C07273=1019.893,90.368,388.919,167.159,51.972,159.571
C07274=1019.887,90.119,388.936,167.157,51.979,159.572
C07275=1019.882,89.870,388.955,167.154,51.985,159.572
C07276=1019.877,89.621,388.972,167.151,51.992,159.573
C07277=1019.872,89.371,388.989,167.149,51.999,159.574
C07278=1019.866,89.122,389.007,167.146,52.005,159.575
C07279=1019.860,88.872,389.025,167.143,52.012,159.575
C07280=1019.855,88.623,389.042,167.141,52.018,159.576
C07281=1019.849,88.374,389.059,167.139,52.025,159.577
C07282=1019.844,88.125,389.077,167.135,52.032,159.578
C07283=1019.838,87.875,389.094,167.133,52.039,159.579
C07284=1019.833,87.626,389.111,167.130,52.046,159.580
C07285=1019.828,87.377,389.129,167.127,52.052,159.580
C07286=1019.821,87.127,389.146,167.124,52.059,159.581
C07287=1019.816,86.877,389.163,167.122,52.065,159.582
C07288=1019.811,86.628,389.181,167.120,52.072,159.583
C07289=1019.805,86.379,389.198,167.116,52.079,159.583
C07290=1019.800,86.130,389.215,167.114,52.085,159.584
C07291=1019.794,85.881,389.233,167.111,52.092,159.585
C07292=1019.789,85.632,389.250,167.108,52.099,159.586
C07293=1019.784,85.382,389.267,167.106,52.106,159.587
C07294=1019.778,85.132,389.285,167.103,52.113,159.587
C07295=1019.772,84.882,389.302,167.100,52.119,159.588
C07296=1019.767,84.633,389.320,167.097,52.126,159.589
C07297=1019.761,84.384,389.337,167.095,52.132,159.590
C07298=1019.756,84.135,389.354,167.093,52.139,159.591
C07299=1019.751,83.886,389.372,167.089,52.145,159.591
C07300=1019.745,83.636,389.388,167.087,52.152,159.592
C07301=1019.739,83.387,389.405,167.085,52.159,159.593
C07302=1019.734,83.138,389.422,167.081,52.166,159.594
C07303=1019.728,82.889,389.440,167.079,52.172,159.594
C07304=1019.723,82.640,389.457,167.076,52.179,159.595
C07305=1019.718,82.390,389.474,167.073,52.185,159.596
C07306=1019.712,82.141,389.492,167.071,52.192,159.597
C07307=1019.706,81.891,389.509,167.068,52.198,159.597
C07308=1019.701,81.641,389.527,167.065,52.205,159.598
C07309=1019.696,81.392,389.543,167.063,52.212,159.599
C07310=1019.690,81.143,389.561,167.060,52.218,159.600
C07311=1019.685,80.893,389.578,167.057,52.225,159.601
C07312=1019.679,80.644,389.595,167.055,52.232,159.602
C07313=1019.674,80.394,389.612,167.052,52.239,159.602
C07314=1019.669,80.145,389.630,167.049,52.245,159.603
C07315=1019.663,79.896,389.647,167.047,52.251,159.604
C07316=1019.658,79.647,389.664,167.044,52.258,159.605
C07317=1019.653,79.397,389.681,167.041,52.264,159.605
C07318=1019.647,79.148,389.699,167.039,52.271,159.606
C07319=1019.641,78.899,389.715,167.036,52.278,159.607
C07320=1019.636,78.650,389.733,167.033,52.284,159.608
C07321=1019.630,78.400,389.749,167.031,52.291,159.608
C07322=1019.625,78.151,389.767,167.028,52.297,159.609
C07323=1019.620,77.901,389.784,167.026,52.304,159.610
C07324=1019.615,77.652,389.801,167.023,52.311,159.611
C07325=1019.609,77.403,389.818,167.021,52.317,159.611
C07326=1019.604,77.153,389.835,167.018,52.324,159.612
C07327=1019.598,76.904,389.853,167.015,52.330,159.613
C07328=1019.592,76.654,389.869,167.013,52.336,159.614
C07329=1019.587,76.405,389.886,167.010,52.343,159.615
C07330=1019.582,76.156,389.903,167.007,52.350,159.615
C07331=1019.576,75.906,389.920,167.004,52.357,159.616
C07332=1019.570,75.657,389.936,167.002,52.363,159.617
C07333=1019.564,75.374,389.955,166.999,52.371,159.618
C07334=1019.558,75.091,389.974,166.996,52.379,159.619
C07335=1019.552,74.810,389.994,166.993,52.386,159.620
C07336=1019.546,74.527,390.013,166.990,52.394,159.621
C07337=1019.541,74.277,390.030,166.987,52.401,159.621
C07338=1019.535,74.027,390.046,166.984,52.407,159.622
C07339=1019.530,73.778,390.063,166.982,52.413,159.623
C07340=1019.524,73.529,390.080,166.979,52.421,159.624
C07341=1019.519,73.279,390.097,166.977,52.427,159.624
C07342=1019.513,73.030,390.113,166.974,52.433,159.625
C07343=1019.508,72.780,390.130,166.971,52.440,159.626
C07344=1019.502,72.531,390.147,166.969,52.447,159.627
C07345=1019.496,72.282,390.164,166.965,52.453,159.627
C07346=1019.491,72.032,390.181,166.963,52.460,159.628
C07347=1019.486,71.783,390.198,166.961,52.467,159.629
C07348=1019.480,71.533,390.214,166.958,52.473,159.630
C07349=1019.475,71.284,390.230,166.955,52.480,159.631
C07350=1019.469,71.035,390.247,166.953,52.487,159.631
C07351=1019.464,70.786,390.264,166.950,52.493,159.632
C07352=1019.458,70.536,390.281,166.948,52.500,159.633
C07353=1019.453,70.287,390.297,166.945,52.507,159.634
C07354=1019.447,70.037,390.314,166.942,52.513,159.634
C07355=1019.442,69.788,390.331,166.940,52.520,159.635
C07356=1019.436,69.538,390.347,166.938,52.526,159.636
C07357=1019.431,69.289,390.364,166.934,52.533,159.637
C07358=1019.426,69.040,390.380,166.932,52.540,159.637
C07359=1019.420,68.790,390.397,166.930,52.546,159.638
C07360=1019.415,68.541,390.414,166.926,52.553,159.639
C07361=1019.409,68.292,390.431,166.924,52.559,159.640
C07362=1019.404,68.042,390.448,166.922,52.566,159.641
C07363=1019.398,67.793,390.464,166.918,52.573,159.641
C07364=1019.393,67.543,390.481,166.916,52.579,159.642
C07365=1019.387,67.295,390.497,166.914,52.586,159.643
C07366=1019.382,67.045,390.513,166.910,52.592,159.644
C07367=1019.376,66.796,390.530,166.908,52.599,159.644
C07368=1019.370,66.546,390.545,166.906,52.606,159.645
C07369=1019.365,66.296,390.562,166.903,52.612,159.646
C07370=1019.359,66.047,390.578,166.900,52.619,159.647
C07371=1019.355,65.798,390.595,166.898,52.626,159.648
C07372=1019.349,65.548,390.611,166.895,52.632,159.648
C07373=1019.343,65.299,390.628,166.893,52.639,159.649
C07374=1019.337,65.049,390.644,166.891,52.646,159.650
C07375=1019.332,64.800,390.661,166.887,52.653,159.651
C07376=1019.326,64.550,390.677,166.885,52.659,159.651
C07377=1019.321,64.302,390.693,166.882,52.666,159.652
C07378=1019.316,64.052,390.710,166.880,52.673,159.653
C07379=1019.310,63.803,390.726,166.877,52.679,159.654
C07380=1019.305,63.552,390.742,166.874,52.686,159.654
C07381=1019.299,63.303,390.759,166.871,52.692,159.655
C07382=1019.294,63.054,390.775,166.869,52.699,159.656
C07383=1019.288,62.805,390.791,166.866,52.706,159.657
C07384=1019.282,62.555,390.808,166.864,52.713,159.658
C07385=1019.277,62.305,390.823,166.860,52.719,159.658
C07386=1019.271,62.056,390.839,166.858,52.726,159.659
C07387=1019.265,61.807,390.855,166.856,52.733,159.660
C07388=1019.260,61.557,390.871,166.853,52.740,159.661
C07389=1019.254,61.308,390.887,166.851,52.746,159.662
C07390=1019.248,61.059,390.903,166.848,52.754,159.662
C07391=1019.243,60.808,390.920,166.845,52.760,159.663
C07392=1019.238,60.560,390.935,166.842,52.767,159.664
C07393=1019.232,60.310,390.952,166.840,52.774,159.665
C07394=1019.226,60.060,390.967,166.838,52.780,159.666
C07395=1019.220,59.811,390.984,166.835,52.787,159.666
C07396=1019.215,59.562,390.999,166.832,52.793,159.667
C07397=1019.208,59.279,391.017,166.830,52.801,159.668
C07398=1019.202,58.996,391.036,166.826,52.810,159.669
C07399=1019.195,58.713,391.054,166.823,52.817,159.670
C07400=1019.189,58.431,391.072,166.820,52.825,159.671
C07401=1019.184,58.181,391.088,166.818,52.831,159.672
C07402=1019.178,57.932,391.104,166.815,52.838,159.672
C07403=1019.172,57.682,391.120,166.812,52.845,159.673
C07404=1019.167,57.433,391.136,166.809,52.852,159.674
C07405=1019.161,57.184,391.152,166.807,52.858,159.675
C07406=1019.155,56.934,391.167,166.805,52.865,159.675
C07407=1019.150,56.685,391.183,166.802,52.872,159.676
C07408=1019.144,56.435,391.199,166.800,52.878,159.677
C07409=1019.139,56.186,391.215,166.796,52.885,159.677
C07410=1019.133,55.937,391.230,166.794,52.892,159.678
C07411=1019.128,55.687,391.246,166.792,52.898,159.679
C07412=1019.122,55.438,391.263,166.788,52.905,159.680
C07413=1019.117,55.188,391.278,166.786,52.912,159.681
C07414=1019.111,54.939,391.295,166.784,52.918,159.682
C07415=1019.106,54.689,391.310,166.781,52.925,159.682
C07416=1019.100,54.440,391.326,166.779,52.932,159.683
C07417=1019.095,54.190,391.342,166.775,52.939,159.684
C07418=1019.089,53.941,391.358,166.773,52.945,159.684
C07419=1019.084,53.692,391.373,166.771,52.952,159.685
C07420=1019.078,53.442,391.389,166.768,52.959,159.686
C07421=1019.072,53.193,391.405,166.765,52.965,159.687
C07422=1019.067,52.944,391.421,166.763,52.972,159.688
C07423=1019.061,52.694,391.436,166.760,52.979,159.688
C07424=1019.056,52.444,391.453,166.758,52.985,159.689
C07425=1019.051,52.195,391.468,166.755,52.992,159.690
C07426=1019.045,51.946,391.485,166.752,52.998,159.690
C07427=1019.039,51.696,391.500,166.750,53.005,159.691
C07428=1019.034,51.447,391.516,166.747,53.012,159.692
C07429=1019.028,51.197,391.532,166.744,53.018,159.693
C07430=1019.023,50.948,391.547,166.742,53.025,159.694
C07431=1019.017,50.698,391.563,166.739,53.032,159.694
C07432=1019.012,50.448,391.579,166.737,53.038,159.695
C07433=1019.006,50.200,391.594,166.735,53.045,159.696
C07434=1019.001,49.950,391.610,166.731,53.052,159.697
C07435=1018.995,49.701,391.626,166.729,53.058,159.697
C07436=1018.990,49.451,391.641,166.727,53.064,159.698
C07437=1018.985,49.201,391.658,166.724,53.072,159.699
C07438=1018.979,48.952,391.673,166.721,53.078,159.700
C07439=1018.974,48.702,391.689,166.719,53.085,159.700
C07440=1018.968,48.454,391.705,166.715,53.091,159.701
C07441=1018.963,48.204,391.720,166.713,53.098,159.702
C07442=1018.958,47.954,391.736,166.711,53.104,159.703
C07443=1018.952,47.705,391.752,166.708,53.111,159.703
C07444=1018.947,47.456,391.767,166.705,53.117,159.704
C07445=1018.941,47.206,391.783,166.703,53.124,159.705
C07446=1018.935,46.957,391.799,166.701,53.130,159.706
C07447=1018.930,46.707,391.814,166.698,53.137,159.706
C07448=1018.924,46.457,391.830,166.695,53.143,159.707
C07449=1018.919,46.209,391.845,166.693,53.150,159.708
C07450=1018.913,45.959,391.861,166.690,53.157,159.708
C07451=1018.908,45.709,391.876,166.688,53.164,159.709
C07452=1018.903,45.460,391.893,166.685,53.170,159.710
C07453=1018.898,45.210,391.908,166.682,53.177,159.711
C07454=1018.892,44.961,391.924,166.680,53.183,159.711
C07455=1018.887,44.712,391.940,166.678,53.190,159.712
C07456=1018.881,44.462,391.955,166.675,53.196,159.713
C07457=1018.876,44.213,391.970,166.672,53.202,159.713
C07458=1018.870,43.963,391.987,166.670,53.209,159.714
C07459=1018.865,43.714,392.002,166.667,53.215,159.715
C07460=1018.860,43.464,392.017,166.664,53.222,159.716
C07461=1018.854,43.182,392.035,166.661,53.230,159.717
C07462=1018.848,42.898,392.053,166.658,53.237,159.717
C07463=1018.842,42.616,392.070,166.655,53.244,159.718
C07464=1018.835,42.333,392.088,166.653,53.252,159.719
C07465=1018.830,42.083,392.103,166.650,53.258,159.720
C07466=1018.824,41.833,392.119,166.648,53.265,159.721
C07467=1018.819,41.584,392.134,166.644,53.271,159.721
C07468=1018.814,41.335,392.148,166.642,53.278,159.722
C07469=1018.808,41.085,392.164,166.640,53.284,159.723
C07470=1018.803,40.836,392.180,166.637,53.292,159.723
C07471=1018.797,40.586,392.195,166.635,53.298,159.724
C07472=1018.792,40.337,392.210,166.632,53.305,159.725
C07473=1018.786,40.088,392.225,166.629,53.312,159.726
C07474=1018.781,39.838,392.241,166.627,53.318,159.726
C07475=1018.775,39.588,392.256,166.624,53.325,159.727
C07476=1018.770,39.339,392.271,166.621,53.331,159.728
C07477=1018.763,39.089,392.286,166.619,53.338,159.729
C07478=1018.758,38.840,392.301,166.616,53.345,159.729
C07479=1018.753,38.591,392.317,166.614,53.351,159.730
C07480=1018.748,38.341,392.332,166.611,53.358,159.731
C07481=1018.742,38.092,392.347,166.608,53.365,159.732
C07482=1018.736,37.842,392.362,166.606,53.371,159.732
C07483=1018.731,37.593,392.377,166.604,53.378,159.733
C07484=1018.726,37.343,392.393,166.600,53.384,159.734
C07485=1018.721,37.093,392.408,166.598,53.391,159.735
C07486=1018.715,36.845,392.423,166.596,53.397,159.735
C07487=1018.709,36.595,392.438,166.593,53.404,159.736
C07488=1018.704,36.345,392.453,166.591,53.411,159.737
C07489=1018.698,36.096,392.468,166.587,53.418,159.738
C07490=1018.693,35.846,392.483,166.585,53.424,159.738
C07491=1018.687,35.597,392.497,166.583,53.431,159.739
C07492=1018.682,35.347,392.513,166.580,53.437,159.740
C07493=1018.676,35.098,392.528,166.578,53.444,159.741
C07494=1018.671,34.849,392.543,166.575,53.451,159.741
C07495=1018.664,34.599,392.558,166.572,53.458,159.742
C07496=1018.660,34.349,392.572,166.569,53.465,159.743
C07497=1018.653,34.099,392.587,166.567,53.471,159.743
C07498=1018.648,33.850,392.602,166.565,53.478,159.744
C07499=1018.642,33.601,392.617,166.561,53.484,159.745
C07500=1018.637,33.351,392.632,166.559,53.491,159.746
C07501=1018.631,33.102,392.646,166.556,53.498,159.746
C07502=1018.626,32.852,392.661,166.554,53.504,159.747
C07503=1018.620,32.603,392.676,166.552,53.511,159.748
C07504=1018.615,32.353,392.691,166.548,53.518,159.749
C07505=1018.609,32.104,392.705,166.546,53.525,159.749
C07506=1018.604,31.854,392.721,166.543,53.531,159.750
C07507=1018.598,31.605,392.735,166.541,53.538,159.751
C07508=1018.593,31.356,392.751,166.538,53.544,159.752
C07509=1018.588,31.105,392.765,166.535,53.552,159.752
C07510=1018.582,30.856,392.780,166.533,53.558,159.753
C07511=1018.577,30.607,392.795,166.530,53.565,159.754
C07512=1018.570,30.357,392.810,166.528,53.571,159.754
C07513=1018.566,30.107,392.825,166.525,53.577,159.755
C07514=1018.560,29.858,392.839,166.522,53.584,159.756
C07515=1018.555,29.609,392.854,166.520,53.591,159.757
C07516=1018.549,29.359,392.869,166.518,53.598,159.757
C07517=1018.544,29.110,392.884,166.514,53.604,159.758
C07518=1018.538,28.861,392.898,166.512,53.611,159.759
C07519=1018.532,28.610,392.913,166.509,53.617,159.759
C07520=1018.527,28.361,392.928,166.507,53.624,159.760
C07521=1018.522,28.112,392.943,166.505,53.630,159.761
C07522=1018.516,27.862,392.957,166.501,53.637,159.761
C07523=1018.511,27.612,392.972,166.499,53.644,159.762
C07524=1018.505,27.363,392.987,166.497,53.650,159.763
C07525=1018.499,27.089,393.003,166.494,53.658,159.764
C07526=1018.492,26.814,393.019,166.491,53.665,159.765
C07527=1018.486,26.539,393.035,166.488,53.673,159.766
C07528=1018.480,26.265,393.051,166.485,53.680,159.766
C07529=1018.475,26.007,393.065,166.482,53.687,159.767
C07530=1018.469,25.749,393.081,166.479,53.694,159.768
C07531=1018.463,25.491,393.096,166.477,53.701,159.769
C07532=1018.457,25.233,393.110,166.474,53.708,159.769
C07533=1018.452,24.984,393.125,166.471,53.714,159.770
C07534=1018.447,24.734,393.139,166.468,53.721,159.771
C07535=1018.441,24.485,393.154,166.466,53.727,159.771
C07536=1018.435,24.235,393.168,166.463,53.735,159.772
C07537=1018.430,23.985,393.183,166.461,53.741,159.773
C07538=1018.424,23.736,393.197,166.459,53.748,159.774
C07539=1018.419,23.487,393.212,166.455,53.754,159.774
C07540=1018.413,23.237,393.226,166.453,53.761,159.775
C07541=1018.408,22.987,393.240,166.450,53.768,159.776
C07542=1018.402,22.738,393.255,166.448,53.775,159.777
C07543=1018.397,22.488,393.269,166.444,53.781,159.777
C07544=1018.391,22.239,393.283,166.443,53.788,159.778
C07545=1018.386,21.989,393.298,166.440,53.794,159.779
C07546=1018.380,21.739,393.312,166.437,53.802,159.779
C07547=1018.374,21.490,393.327,166.435,53.808,159.780
C07548=1018.369,21.241,393.341,166.431,53.814,159.781
C07549=1018.364,20.991,393.356,166.429,53.821,159.782
C07550=1018.358,20.742,393.370,166.427,53.827,159.782
C07551=1018.353,20.492,393.384,166.424,53.835,159.783
C07552=1018.347,20.243,393.398,166.422,53.841,159.784
C07553=1018.342,19.993,393.413,166.419,53.848,159.784
C07554=1018.336,19.743,393.427,166.416,53.854,159.785
C07555=1018.330,19.494,393.441,166.414,53.860,159.786
C07556=1018.325,19.245,393.455,166.411,53.868,159.786
C07557=1018.320,18.995,393.470,166.409,53.874,159.787
C07558=1018.314,18.746,393.484,166.406,53.881,159.788
C07559=1018.309,18.496,393.498,166.403,53.887,159.789
C07560=1018.303,18.246,393.512,166.400,53.894,159.789
C07561=1018.297,17.996,393.526,166.398,53.901,159.790
C07562=1018.292,17.747,393.541,166.394,53.908,159.791
C07563=1018.286,17.498,393.555,166.393,53.914,159.791
C07564=1018.281,17.248,393.569,166.390,53.921,159.792
C07565=1018.275,16.999,393.582,166.387,53.928,159.793
C07566=1018.269,16.750,393.597,166.385,53.934,159.794
C07567=1018.265,16.500,393.611,166.382,53.941,159.794
C07568=1018.259,16.250,393.625,166.380,53.948,159.795
C07569=1018.254,16.001,393.639,166.376,53.954,159.795
C07570=1018.248,15.751,393.653,166.374,53.961,159.796
C07571=1018.242,15.501,393.667,166.371,53.968,159.797
C07572=1018.236,15.252,393.682,166.369,53.975,159.798
C07573=1018.231,15.002,393.696,166.367,53.981,159.798
C07574=1018.225,14.753,393.710,166.363,53.987,159.799
C07575=1018.220,14.503,393.723,166.361,53.994,159.800
C07576=1018.214,14.253,393.737,166.358,54.001,159.800
C07577=1018.209,14.004,393.751,166.355,54.007,159.801
C07578=1018.204,13.755,393.766,166.352,54.014,159.802
C07579=1018.198,13.505,393.780,166.350,54.021,159.803
C07580=1018.193,13.255,393.794,166.348,54.027,159.803
C07581=1018.187,13.006,393.808,166.345,54.034,159.804
C07582=1018.181,12.757,393.821,166.343,54.041,159.805
C07583=1018.176,12.507,393.835,166.339,54.048,159.805
C07584=1018.170,12.258,393.849,166.337,54.055,159.806
C07585=1018.165,12.008,393.863,166.334,54.061,159.807
C07586=1018.159,11.758,393.877,166.331,54.069,159.808
C07587=1018.153,11.509,393.890,166.329,54.075,159.808
C07588=1018.148,11.259,393.903,166.326,54.082,159.809
C07589=1018.142,10.977,393.919,166.323,54.089,159.810
C07590=1018.135,10.696,393.934,166.320,54.097,159.811
C07591=1018.129,10.415,393.950,166.318,54.105,159.812
C07592=1018.123,10.133,393.965,166.314,54.112,159.812
C07593=1018.117,9.884,393.979,166.311,54.119,159.813
C07594=1018.111,9.634,393.993,166.308,54.126,159.814
C07595=1018.106,9.385,394.006,166.306,54.132,159.814
C07596=1018.100,9.135,394.020,166.303,54.140,159.815
C07597=1018.095,8.886,394.034,166.301,54.146,159.816
C07598=1018.090,8.636,394.047,166.298,54.153,159.816
C07599=1018.083,8.386,394.061,166.296,54.159,159.817
C07600=1018.078,8.137,394.074,166.293,54.167,159.818
C07601=1018.073,7.887,394.088,166.290,54.173,159.819
C07602=1018.067,7.638,394.102,166.287,54.179,159.819
C07603=1018.061,7.388,394.115,166.285,54.186,159.820
C07604=1018.056,7.138,394.129,166.282,54.193,159.820
C07605=1018.050,6.888,394.142,166.280,54.200,159.821
C07606=1018.045,6.639,394.156,166.276,54.207,159.822
C07607=1018.039,6.389,394.170,166.274,54.213,159.823
C07608=1018.034,6.141,394.183,166.271,54.220,159.823
C07609=1018.028,5.891,394.197,166.269,54.226,159.824
C07610=1018.023,5.641,394.210,166.265,54.233,159.825
C07611=1018.017,5.391,394.224,166.264,54.240,159.825
C07612=1018.012,5.142,394.238,166.260,54.247,159.826
C07613=1018.006,4.893,394.251,166.258,54.253,159.827
C07614=1018.000,4.643,394.265,166.255,54.260,159.827
C07615=1017.995,4.393,394.278,166.253,54.266,159.828
C07616=1017.990,4.143,394.292,166.250,54.273,159.829
C07617=1017.984,3.894,394.306,166.247,54.280,159.829
C07618=1017.979,3.645,394.319,166.245,54.286,159.830
C07619=1017.973,3.395,394.332,166.242,54.293,159.831
C07620=1017.968,3.145,394.346,166.240,54.300,159.832
C07621=1017.962,2.896,394.360,166.236,54.306,159.832
C07622=1017.957,2.646,394.372,166.234,54.313,159.833
C07623=1017.951,2.396,394.386,166.231,54.320,159.834
C07624=1017.946,2.147,394.400,166.229,54.326,159.834
C07625=1017.941,1.898,394.413,166.225,54.333,159.835
C07626=1017.936,1.648,394.427,166.223,54.339,159.835
C07627=1017.929,1.398,394.440,166.220,54.346,159.836
C07628=1017.924,1.149,394.454,166.218,54.353,159.837
C07629=1017.919,0.899,394.467,166.215,54.359,159.837
C07630=1017.913,0.649,394.481,166.212,54.366,159.838
C07631=1017.908,0.401,394.494,166.210,54.373,159.839
C07632=1017.902,0.150,394.507,166.207,54.379,159.839
C07633=1017.897,-0.099,394.521,166.205,54.385,159.840
C07634=1017.891,-0.349,394.534,166.201,54.392,159.841
C07635=1017.886,-0.599,394.548,166.199,54.398,159.841
C07636=1017.881,-0.848,394.561,166.196,54.406,159.842
C07637=1017.875,-1.097,394.574,166.194,54.412,159.843
C07638=1017.870,-1.347,394.588,166.192,54.418,159.843
C07639=1017.865,-1.597,394.601,166.188,54.425,159.844
C07640=1017.859,-1.846,394.614,166.186,54.431,159.845
C07641=1017.854,-2.096,394.627,166.183,54.438,159.845
C07642=1017.848,-2.345,394.641,166.181,54.445,159.846
C07643=1017.843,-2.595,394.654,166.177,54.451,159.847
C07644=1017.838,-2.844,394.667,166.175,54.458,159.847
C07645=1017.832,-3.094,394.680,166.173,54.464,159.848
C07646=1017.827,-3.344,394.694,166.169,54.471,159.848
C07647=1017.822,-3.594,394.708,166.167,54.477,159.849
C07648=1017.817,-3.843,394.721,166.164,54.484,159.850
C07649=1017.811,-4.092,394.734,166.162,54.490,159.850
C07650=1017.805,-4.342,394.747,166.158,54.497,159.851
C07651=1017.800,-4.593,394.761,166.156,54.503,159.852
C07652=1017.794,-4.842,394.774,166.153,54.510,159.852
C07653=1017.788,-5.121,394.788,166.150,54.518,159.853
C07654=1017.782,-5.400,394.803,166.148,54.525,159.854
C07655=1017.776,-5.680,394.817,166.145,54.533,159.855
C07656=1017.770,-5.959,394.831,166.141,54.541,159.855
C07657=1017.764,-6.209,394.844,166.139,54.547,159.856
C07658=1017.758,-6.459,394.857,166.136,54.554,159.857
C07659=1017.753,-6.709,394.870,166.133,54.561,159.857
C07660=1017.748,-6.958,394.883,166.130,54.567,159.858
C07661=1017.742,-7.208,394.896,166.128,54.574,159.859
C07662=1017.736,-7.457,394.909,166.125,54.581,159.859
C07663=1017.731,-7.706,394.922,166.122,54.588,159.860
C07664=1017.725,-7.956,394.935,166.119,54.594,159.861
C07665=1017.720,-8.206,394.948,166.116,54.601,159.861
C07666=1017.715,-8.456,394.960,166.114,54.607,159.862
C07667=1017.708,-8.705,394.973,166.111,54.614,159.862
C07668=1017.703,-8.955,394.986,166.109,54.621,159.863
C07669=1017.698,-9.204,394.999,166.106,54.628,159.864
C07670=1017.693,-9.454,395.012,166.103,54.634,159.865
C07671=1017.687,-9.704,395.025,166.100,54.641,159.865
C07672=1017.681,-9.953,395.037,166.098,54.648,159.866
C07673=1017.676,-10.203,395.050,166.095,54.654,159.867
C07674=1017.671,-10.452,395.063,166.093,54.661,159.867
C07675=1017.666,-10.702,395.076,166.089,54.667,159.868
C07676=1017.659,-10.952,395.089,166.086,54.675,159.868
C07677=1017.654,-11.201,395.101,166.084,54.681,159.869
C07678=1017.649,-11.451,395.114,166.081,54.688,159.870
C07679=1017.643,-11.701,395.127,166.079,54.694,159.870
C07680=1017.638,-11.950,395.140,166.075,54.701,159.871
C07681=1017.632,-12.200,395.153,166.073,54.707,159.871
C07682=1017.627,-12.449,395.165,166.070,54.714,159.872
C07683=1017.622,-12.699,395.178,166.068,54.721,159.873
C07684=1017.616,-12.949,395.191,166.064,54.727,159.873
C07685=1017.611,-13.198,395.203,166.062,54.734,159.874
C07686=1017.605,-13.448,395.216,166.059,54.740,159.875
C07687=1017.600,-13.698,395.228,166.057,54.747,159.875
C07688=1017.595,-13.947,395.242,166.054,54.754,159.876
C07689=1017.589,-14.196,395.254,166.052,54.760,159.877
C07690=1017.583,-14.446,395.267,166.048,54.767,159.877
C07691=1017.579,-14.696,395.280,166.046,54.773,159.878
C07692=1017.573,-14.946,395.292,166.043,54.780,159.878
C07693=1017.567,-15.195,395.305,166.040,54.786,159.879
C07694=1017.562,-15.445,395.318,166.037,54.793,159.880
C07695=1017.556,-15.695,395.330,166.035,54.799,159.880
C07696=1017.552,-15.944,395.343,166.031,54.806,159.881
C07697=1017.546,-16.194,395.355,166.030,54.813,159.882
C07698=1017.541,-16.443,395.368,166.026,54.820,159.882
C07699=1017.535,-16.693,395.380,166.024,54.826,159.883
C07700=1017.529,-16.942,395.392,166.021,54.833,159.883
C07701=1017.524,-17.192,395.405,166.018,54.840,159.884
C07702=1017.518,-17.442,395.417,166.016,54.846,159.885
C07703=1017.512,-17.691,395.430,166.012,54.853,159.885
C07704=1017.508,-17.941,395.442,166.010,54.859,159.886
C07705=1017.502,-18.191,395.455,166.007,54.867,159.887
C07706=1017.497,-18.441,395.466,166.004,54.874,159.887
C07707=1017.491,-18.690,395.479,166.002,54.880,159.888
C07708=1017.486,-18.940,395.491,165.998,54.887,159.888
C07709=1017.480,-19.190,395.504,165.997,54.894,159.889
C07710=1017.474,-19.439,395.516,165.993,54.900,159.890
C07711=1017.469,-19.689,395.529,165.990,54.907,159.890
C07712=1017.463,-19.938,395.541,165.988,54.913,159.891
C07713=1017.458,-20.188,395.553,165.985,54.920,159.892
C07714=1017.453,-20.438,395.565,165.983,54.927,159.892
C07715=1017.447,-20.688,395.578,165.979,54.934,159.893
C07716=1017.442,-20.937,395.590,165.977,54.940,159.894
C07717=1017.436,-21.214,395.603,165.973,54.948,159.894
C07718=1017.430,-21.491,395.617,165.971,54.955,159.895
C07719=1017.424,-21.770,395.631,165.967,54.962,159.896
C07720=1017.418,-22.048,395.644,165.965,54.970,159.896
C07721=1017.412,-22.297,395.656,165.961,54.976,159.897
C07722=1017.406,-22.547,395.669,165.959,54.983,159.897
C07723=1017.401,-22.796,395.681,165.956,54.990,159.898
C07724=1017.396,-23.047,395.693,165.954,54.996,159.899
C07725=1017.390,-23.296,395.705,165.951,55.003,159.899
C07726=1017.386,-23.545,395.718,165.947,55.010,159.900
C07727=1017.380,-23.795,395.730,165.945,55.016,159.901
C07728=1017.375,-24.045,395.742,165.942,55.023,159.901
C07729=1017.369,-24.294,395.754,165.940,55.029,159.902
C07730=1017.364,-24.544,395.767,165.936,55.036,159.902
C07731=1017.359,-24.794,395.778,165.934,55.042,159.903
C07732=1017.353,-25.044,395.791,165.931,55.049,159.903
C07733=1017.347,-25.293,395.803,165.929,55.055,159.904
C07734=1017.342,-25.542,395.815,165.925,55.062,159.905
C07735=1017.336,-25.792,395.827,165.923,55.068,159.905
C07736=1017.331,-26.042,395.839,165.920,55.075,159.906
C07737=1017.326,-26.291,395.851,165.918,55.081,159.906
C07738=1017.321,-26.542,395.864,165.914,55.088,159.907
C07739=1017.316,-26.791,395.876,165.911,55.095,159.907
C07740=1017.310,-27.040,395.888,165.909,55.101,159.908
C07741=1017.305,-27.291,395.900,165.905,55.108,159.909
C07742=1017.299,-27.540,395.912,165.903,55.114,159.909
C07743=1017.294,-27.790,395.924,165.900,55.122,159.910
C07744=1017.288,-28.039,395.936,165.898,55.128,159.911
C07745=1017.283,-28.289,395.948,165.895,55.135,159.911
C07746=1017.277,-28.538,395.959,165.892,55.141,159.912
C07747=1017.272,-28.789,395.971,165.889,55.148,159.912
C07748=1017.267,-29.038,395.983,165.886,55.155,159.913
C07749=1017.262,-29.288,395.995,165.884,55.162,159.914
C07750=1017.257,-29.537,396.006,165.881,55.168,159.914
C07751=1017.250,-29.787,396.018,165.878,55.175,159.915
C07752=1017.245,-30.037,396.030,165.876,55.181,159.916
C07753=1017.240,-30.286,396.042,165.872,55.188,159.916
C07754=1017.234,-30.536,396.054,165.869,55.195,159.917
C07755=1017.229,-30.786,396.066,165.867,55.201,159.917
C07756=1017.223,-31.035,396.077,165.864,55.208,159.918
C07757=1017.218,-31.285,396.088,165.862,55.215,159.919
C07758=1017.212,-31.535,396.101,165.859,55.222,159.919
C07759=1017.207,-31.785,396.112,165.855,55.229,159.920
C07760=1017.202,-32.034,396.124,165.853,55.235,159.920
C07761=1017.196,-32.283,396.135,165.850,55.242,159.921
C07762=1017.191,-32.533,396.147,165.847,55.248,159.921
C07763=1017.185,-32.783,396.159,165.845,55.255,159.922
C07764=1017.180,-33.033,396.171,165.841,55.261,159.923
C07765=1017.175,-33.283,396.182,165.839,55.268,159.923
C07766=1017.169,-33.531,396.194,165.836,55.275,159.924
C07767=1017.164,-33.781,396.205,165.833,55.281,159.924
C07768=1017.158,-34.032,396.217,165.830,55.288,159.925
C07769=1017.153,-34.281,396.229,165.827,55.294,159.925
C07770=1017.147,-34.530,396.240,165.825,55.301,159.926
C07771=1017.142,-34.780,396.252,165.822,55.308,159.927
C07772=1017.137,-35.029,396.264,165.819,55.314,159.927
C07773=1017.131,-35.280,396.276,165.816,55.321,159.928
C07774=1017.126,-35.530,396.287,165.813,55.327,159.928
C07775=1017.121,-35.779,396.298,165.811,55.334,159.929
C07776=1017.115,-36.028,396.310,165.807,55.341,159.929
C07777=1017.110,-36.278,396.322,165.805,55.347,159.930
C07778=1017.105,-36.528,396.333,165.802,55.354,159.931
C07779=1017.100,-36.778,396.345,165.800,55.360,159.931
C07780=1017.094,-37.027,396.357,165.797,55.367,159.932
C07781=1017.088,-37.304,396.369,165.794,55.374,159.933
C07782=1017.083,-37.581,396.382,165.791,55.381,159.933
C07783=1017.076,-37.857,396.395,165.787,55.389,159.934
C07784=1017.071,-38.134,396.408,165.784,55.396,159.934
C07785=1017.066,-38.384,396.419,165.781,55.402,159.935
C07786=1017.060,-38.633,396.431,165.778,55.409,159.935
C07787=1017.055,-38.882,396.442,165.776,55.415,159.936
C07788=1017.050,-39.132,396.454,165.773,55.422,159.936
C07789=1017.044,-39.383,396.465,165.771,55.428,159.937
C07790=1017.039,-39.632,396.476,165.767,55.435,159.938
C07791=1017.034,-39.882,396.488,165.764,55.442,159.938
C07792=1017.028,-40.132,396.499,165.762,55.448,159.939
C07793=1017.023,-40.381,396.510,165.759,55.455,159.939
C07794=1017.017,-40.631,396.521,165.755,55.462,159.940
C07795=1017.012,-40.881,396.532,165.753,55.468,159.940
C07796=1017.006,-41.130,396.543,165.750,55.475,159.941
C07797=1017.001,-41.380,396.555,165.747,55.482,159.941
C07798=1016.996,-41.629,396.566,165.745,55.488,159.942
C07799=1016.991,-41.879,396.577,165.741,55.495,159.943
C07800=1016.985,-42.129,396.588,165.738,55.502,159.943
C07801=1016.980,-42.379,396.599,165.736,55.508,159.944
C07802=1016.974,-42.628,396.610,165.733,55.515,159.944
C07803=1016.969,-42.878,396.622,165.729,55.522,159.945
C07804=1016.963,-43.127,396.633,165.727,55.528,159.945
C07805=1016.958,-43.377,396.644,165.724,55.535,159.946
C07806=1016.953,-43.627,396.655,165.722,55.541,159.947
C07807=1016.948,-43.876,396.667,165.719,55.548,159.947
C07808=1016.942,-44.126,396.677,165.715,55.555,159.948
C07809=1016.937,-44.376,396.689,165.713,55.561,159.948
C07810=1016.932,-44.626,396.699,165.710,55.568,159.949
C07811=1016.927,-44.876,396.710,165.707,55.575,159.949
C07812=1016.921,-45.125,396.721,165.705,55.581,159.950
C07813=1016.916,-45.375,396.733,165.701,55.588,159.950
C07814=1016.910,-45.624,396.744,165.699,55.594,159.951
C07815=1016.905,-45.874,396.755,165.696,55.601,159.952
C07816=1016.899,-46.124,396.766,165.693,55.608,159.952
C07817=1016.894,-46.373,396.778,165.691,55.614,159.953
C07818=1016.889,-46.624,396.788,165.687,55.621,159.953
C07819=1016.884,-46.873,396.799,165.685,55.627,159.954
C07820=1016.878,-47.123,396.810,165.682,55.634,159.954
C07821=1016.873,-47.373,396.822,165.678,55.640,159.955
C07822=1016.867,-47.622,396.832,165.676,55.647,159.955
C07823=1016.863,-47.873,396.843,165.673,55.654,159.956
C07824=1016.857,-48.122,396.854,165.671,55.660,159.957
C07825=1016.853,-48.371,396.865,165.668,55.667,159.957
C07826=1016.847,-48.621,396.876,165.665,55.673,159.958
C07827=1016.842,-48.870,396.887,165.662,55.679,159.958
C07828=1016.836,-49.121,396.898,165.659,55.686,159.958
C07829=1016.831,-49.370,396.909,165.656,55.692,159.959
C07830=1016.826,-49.620,396.920,165.653,55.699,159.960
C07831=1016.820,-49.869,396.931,165.651,55.706,159.960
C07832=1016.815,-50.120,396.942,165.647,55.712,159.961
C07833=1016.810,-50.369,396.953,165.645,55.718,159.961
C07834=1016.805,-50.619,396.964,165.642,55.725,159.962
C07835=1016.800,-50.870,396.975,165.639,55.732,159.962
C07836=1016.795,-51.118,396.985,165.637,55.738,159.963
C07837=1016.789,-51.368,396.996,165.633,55.745,159.963
C07838=1016.784,-51.618,397.006,165.630,55.752,159.964
C07839=1016.778,-51.867,397.017,165.628,55.758,159.965
C07840=1016.772,-52.118,397.027,165.625,55.765,159.965
C07841=1016.767,-52.367,397.038,165.622,55.772,159.966
C07842=1016.761,-52.617,397.048,165.618,55.779,159.966
C07843=1016.757,-52.866,397.059,165.616,55.785,159.967
C07844=1016.751,-53.116,397.070,165.613,55.792,159.967
C07845=1016.745,-53.394,397.081,165.610,55.799,159.968
C07846=1016.739,-53.670,397.093,165.606,55.807,159.968
C07847=1016.733,-53.947,397.104,165.603,55.814,159.969
C07848=1016.727,-54.224,397.115,165.601,55.822,159.970
C07849=1016.721,-54.474,397.126,165.598,55.829,159.970
C07850=1016.716,-54.724,397.137,165.594,55.835,159.971
C07851=1016.711,-54.973,397.148,165.591,55.842,159.971
C07852=1016.706,-55.223,397.158,165.589,55.849,159.972
C07853=1016.700,-55.473,397.168,165.586,55.855,159.972
C07854=1016.695,-55.723,397.179,165.583,55.862,159.973
C07855=1016.689,-55.973,397.189,165.581,55.869,159.974
C07856=1016.684,-56.222,397.199,165.577,55.876,159.974
C07857=1016.679,-56.472,397.210,165.574,55.882,159.975
C07858=1016.673,-56.722,397.220,165.571,55.889,159.975
C07859=1016.668,-56.971,397.231,165.568,55.895,159.975
C07860=1016.663,-57.221,397.240,165.565,55.902,159.976
C07861=1016.657,-57.471,397.251,165.562,55.909,159.976
C07862=1016.652,-57.720,397.261,165.560,55.915,159.977
C07863=1016.647,-57.970,397.271,165.557,55.922,159.978
C07864=1016.641,-58.220,397.281,165.554,55.929,159.978
C07865=1016.636,-58.470,397.293,165.551,55.935,159.979
C07866=1016.631,-58.720,397.303,165.548,55.942,159.979
C07867=1016.626,-58.969,397.313,165.545,55.949,159.980
C07868=1016.621,-59.219,397.323,165.543,55.955,159.980
C07869=1016.615,-59.469,397.334,165.539,55.961,159.981
C07870=1016.610,-59.718,397.344,165.536,55.968,159.981
C07871=1016.605,-59.968,397.354,165.534,55.975,159.982
C07872=1016.599,-60.218,397.365,165.531,55.981,159.982
C07873=1016.594,-60.467,397.374,165.528,55.988,159.983
C07874=1016.589,-60.717,397.385,165.525,55.995,159.984
C07875=1016.583,-60.967,397.395,165.522,56.001,159.984
C07876=1016.578,-61.216,397.405,165.520,56.007,159.984
C07877=1016.573,-61.466,397.415,165.517,56.014,159.985
C07878=1016.568,-61.716,397.425,165.513,56.021,159.985
C07879=1016.562,-61.966,397.435,165.511,56.027,159.986
C07880=1016.557,-62.216,397.446,165.508,56.033,159.986
C07881=1016.552,-62.465,397.456,165.504,56.040,159.987
C07882=1016.546,-62.715,397.466,165.502,56.047,159.987
C07883=1016.541,-62.965,397.476,165.499,56.054,159.988
C07884=1016.537,-63.215,397.487,165.496,56.059,159.988
C07885=1016.531,-63.465,397.497,165.493,56.066,159.989
C07886=1016.527,-63.714,397.507,165.490,56.073,159.989
C07887=1016.521,-63.964,397.518,165.488,56.079,159.990
C07888=1016.515,-64.214,397.528,165.484,56.086,159.990
C07889=1016.511,-64.463,397.538,165.481,56.092,159.991
C07890=1016.505,-64.713,397.548,165.479,56.099,159.991
C07891=1016.500,-64.963,397.558,165.476,56.106,159.992
C07892=1016.495,-65.213,397.568,165.473,56.111,159.992
C07893=1016.490,-65.462,397.578,165.470,56.118,159.993
C07894=1016.484,-65.712,397.588,165.468,56.125,159.993
C07895=1016.479,-65.961,397.598,165.464,56.131,159.994
C07896=1016.474,-66.211,397.608,165.461,56.138,159.994
C07897=1016.469,-66.461,397.618,165.459,56.144,159.995
C07898=1016.464,-66.711,397.628,165.455,56.150,159.995
C07899=1016.458,-66.961,397.638,165.453,56.157,159.996
C07900=1016.453,-67.210,397.648,165.450,56.164,159.996
C07901=1016.448,-67.460,397.658,165.448,56.169,159.997
C07902=1016.443,-67.710,397.668,165.444,56.176,159.997
C07903=1016.438,-67.960,397.678,165.441,56.182,159.997
C07904=1016.433,-68.209,397.688,165.439,56.189,159.998
C07905=1016.428,-68.459,397.698,165.435,56.196,159.998
C07906=1016.423,-68.709,397.708,165.433,56.201,159.999
C07907=1016.418,-68.958,397.718,165.430,56.208,159.999
C07908=1016.412,-69.208,397.728,165.427,56.214,160.000
C07909=1016.408,-69.486,397.739,165.424,56.222,160.001
C07910=1016.401,-69.764,397.751,165.420,56.229,160.001
C07911=1016.396,-70.042,397.762,165.417,56.236,160.001
C07912=1016.389,-70.321,397.773,165.414,56.243,160.002
C07913=1016.385,-70.570,397.783,165.412,56.249,160.002
C07914=1016.380,-70.820,397.792,165.408,56.255,160.003
C07915=1016.374,-71.070,397.803,165.405,56.262,160.003
C07916=1016.370,-71.319,397.812,165.402,56.268,160.004
C07917=1016.364,-71.569,397.823,165.399,56.275,160.004
C07918=1016.359,-71.819,397.832,165.397,56.280,160.004
C07919=1016.354,-72.069,397.842,165.394,56.287,160.005
C07920=1016.349,-72.319,397.852,165.391,56.293,160.005
C07921=1016.345,-72.568,397.861,165.388,56.300,160.006
C07922=1016.339,-72.818,397.872,165.385,56.306,160.006
C07923=1016.335,-73.068,397.882,165.382,56.313,160.007
C07924=1016.330,-73.317,397.892,165.379,56.318,160.007
C07925=1016.325,-73.568,397.902,165.377,56.324,160.008
C07926=1016.320,-73.817,397.912,165.374,56.331,160.008
C07927=1016.314,-74.067,397.922,165.371,56.337,160.008
C07928=1016.310,-74.317,397.931,165.368,56.344,160.009
C07929=1016.305,-74.567,397.941,165.365,56.349,160.009
C07930=1016.299,-74.816,397.950,165.362,56.356,160.010
C07931=1016.294,-75.066,397.960,165.358,56.362,160.010
C07932=1016.290,-75.316,397.969,165.356,56.369,160.011
C07933=1016.283,-75.566,397.979,165.353,56.376,160.011
C07934=1016.279,-75.815,397.989,165.351,56.381,160.012
C07935=1016.274,-76.065,397.998,165.348,56.388,160.012
C07936=1016.269,-76.315,398.008,165.344,56.395,160.013
C07937=1016.263,-76.564,398.017,165.342,56.401,160.013
C07938=1016.259,-76.814,398.026,165.339,56.408,160.013
C07939=1016.253,-77.064,398.036,165.336,56.414,160.014
C07940=1016.248,-77.314,398.045,165.333,56.420,160.014
C07941=1016.243,-77.563,398.055,165.330,56.427,160.015
C07942=1016.238,-77.814,398.065,165.327,56.433,160.015
C07943=1016.233,-78.064,398.074,165.324,56.440,160.016
C07944=1016.227,-78.313,398.083,165.322,56.446,160.016
C07945=1016.223,-78.563,398.092,165.318,56.453,160.017
C07946=1016.217,-78.813,398.102,165.316,56.458,160.017
C07947=1016.212,-79.062,398.111,165.313,56.465,160.017
C07948=1016.207,-79.312,398.121,165.309,56.471,160.018
C07949=1016.203,-79.561,398.130,165.307,56.478,160.018
C07950=1016.197,-79.812,398.139,165.303,56.484,160.019
C07951=1016.192,-80.061,398.149,165.301,56.491,160.019
C07952=1016.187,-80.311,398.158,165.298,56.497,160.019
C07953=1016.182,-80.560,398.167,165.296,56.503,160.020
C07954=1016.177,-80.811,398.177,165.292,56.510,160.021
C07955=1016.171,-81.061,398.185,165.289,56.517,160.021
C07956=1016.167,-81.310,398.195,165.287,56.523,160.021
C07957=1016.161,-81.560,398.203,165.284,56.530,160.022
C07958=1016.156,-81.809,398.213,165.281,56.537,160.022
C07959=1016.151,-82.060,398.222,165.278,56.542,160.023
C07960=1016.145,-82.309,398.231,165.275,56.549,160.023
C07961=1016.140,-82.559,398.240,165.272,56.556,160.024
C07962=1016.135,-82.809,398.249,165.269,56.562,160.024
C07963=1016.131,-83.059,398.258,165.266,56.569,160.025
C07964=1016.125,-83.309,398.267,165.263,56.576,160.025
C07965=1016.120,-83.558,398.277,165.260,56.582,160.026
C07966=1016.115,-83.808,398.285,165.257,56.589,160.026
C07967=1016.109,-84.058,398.294,165.255,56.594,160.026
C07968=1016.105,-84.307,398.303,165.252,56.601,160.027
C07969=1016.099,-84.557,398.312,165.248,56.608,160.027
C07970=1016.095,-84.807,398.321,165.246,56.614,160.028
C07971=1016.089,-85.057,398.330,165.243,56.621,160.028
C07972=1016.084,-85.307,398.340,165.240,56.627,160.029
C07973=1016.079,-85.587,398.349,165.237,56.635,160.029
C07974=1016.073,-85.867,398.359,165.233,56.642,160.030
C07975=1016.067,-86.147,398.369,165.230,56.648,160.030
C07976=1016.061,-86.426,398.379,165.226,56.656,160.030
C07977=1016.057,-86.676,398.388,165.224,56.662,160.031
C07978=1016.051,-86.927,398.397,165.221,56.669,160.031
///RCONF 1,0,0,0,1,0,0,0,0,0,0,0,0,0,0,0,0,0,0,0,0,0,0,0
C07979=1016.046,-87.176,398.406,165.219,56.675,160.032
C07980=1016.041,-87.426,398.415,165.215,56.681,160.032
C07981=1016.035,-87.675,398.424,165.213,56.688,160.033
C07982=1016.031,-87.925,398.433,165.209,56.694,160.033
C07983=1016.026,-88.175,398.441,165.206,56.701,160.034
C07984=1016.020,-88.425,398.450,165.204,56.707,160.034
C07985=1016.016,-88.675,398.459,165.200,56.714,160.034
C07986=1016.011,-88.925,398.467,165.198,56.719,160.035
C07987=1016.006,-89.175,398.477,165.195,56.726,160.035
C07988=1016.000,-89.424,398.486,165.192,56.732,160.036
C07989=1015.996,-89.674,398.495,165.189,56.738,160.036
C07990=1015.991,-89.924,398.503,165.187,56.745,160.037
C07991=1015.985,-90.173,398.512,165.183,56.751,160.037
C07992=1015.981,-90.423,398.521,165.181,56.757,160.038
C07993=1015.976,-90.673,398.529,165.177,56.764,160.038
C07994=1015.971,-90.923,398.538,165.175,56.770,160.038
C07995=1015.966,-91.173,398.547,165.172,56.776,160.039
C07996=1015.961,-91.422,398.555,165.169,56.782,160.039
C07997=1015.956,-91.672,398.564,165.166,56.789,160.039
C07998=1015.951,-91.922,398.573,165.163,56.795,160.040
C07999=1015.946,-92.172,398.583,165.160,56.801,160.040
C08000=1015.941,-92.421,398.591,165.158,56.808,160.041
C08001=1015.935,-92.671,398.600,165.154,56.814,160.041
C08002=1015.931,-92.921,398.609,165.152,56.820,160.041
C08003=1015.926,-93.171,398.617,165.148,56.827,160.042
C08004=1015.920,-93.420,398.626,165.146,56.832,160.042
C08005=1015.916,-93.671,398.635,165.142,56.839,160.042
C08006=1015.911,-93.920,398.643,165.140,56.845,160.043
C08007=1015.906,-94.170,398.652,165.137,56.851,160.043
C08008=1015.901,-94.420,398.661,165.134,56.857,160.044
C08009=1015.896,-94.670,398.669,165.131,56.864,160.044
C08010=1015.891,-94.920,398.678,165.128,56.870,160.045
C08011=1015.886,-95.169,398.687,165.125,56.876,160.045
C08012=1015.882,-95.419,398.695,165.122,56.882,160.045
C08013=1015.877,-95.669,398.703,165.120,56.888,160.046
C08014=1015.872,-95.919,398.712,165.117,56.895,160.046
C08015=1015.867,-96.169,398.721,165.114,56.900,160.046
C08016=1015.862,-96.419,398.730,165.110,56.907,160.047
C08017=1015.857,-96.669,398.739,165.108,56.913,160.047
C08018=1015.852,-96.918,398.747,165.105,56.919,160.047
C08019=1015.847,-97.167,398.755,165.102,56.925,160.048
C08020=1015.843,-97.417,398.764,165.100,56.931,160.048
C08021=1015.838,-97.667,398.773,165.096,56.937,160.048
C08022=1015.833,-97.917,398.782,165.094,56.944,160.049
C08023=1015.828,-98.167,398.790,165.090,56.950,160.049
C08024=1015.823,-98.417,398.798,165.088,56.956,160.050
C08025=1015.818,-98.667,398.807,165.085,56.963,160.050
C08026=1015.813,-98.916,398.814,165.082,56.969,160.051
C08027=1015.808,-99.166,398.822,165.079,56.975,160.051
C08028=1015.803,-99.416,398.831,165.077,56.981,160.051
C08029=1015.797,-99.666,398.839,165.073,56.987,160.052
C08030=1015.792,-99.916,398.847,165.071,56.994,160.052
C08031=1015.788,-100.166,398.856,165.067,57.000,160.052
C08032=1015.783,-100.415,398.864,165.065,57.006,160.053
C08033=1015.778,-100.665,398.872,165.062,57.013,160.053
C08034=1015.773,-100.915,398.881,165.059,57.019,160.054
C08035=1015.768,-101.165,398.888,165.056,57.025,160.054
C08036=1015.763,-101.414,398.897,165.054,57.032,160.055
C08037=1015.758,-101.697,398.906,165.051,57.039,160.055
C08038=1015.752,-101.978,398.915,165.047,57.046,160.055
C08039=1015.746,-102.261,398.924,165.043,57.052,160.056
C08040=1015.741,-102.543,398.933,165.040,57.059,160.056
C08041=1015.736,-102.793,398.942,165.038,57.066,160.057
C08042=1015.731,-103.042,398.950,165.034,57.072,160.057
C08043=1015.726,-103.293,398.958,165.032,57.078,160.057
C08044=1015.721,-103.542,398.966,165.028,57.084,160.057
C08045=1015.716,-103.792,398.974,165.026,57.091,160.058
C08046=1015.711,-104.042,398.983,165.023,57.097,160.058
C08047=1015.706,-104.292,398.990,165.020,57.103,160.059
C08048=1015.702,-104.541,398.999,165.017,57.108,160.059
C08049=1015.697,-104.792,399.007,165.014,57.115,160.060
C08050=1015.692,-105.042,399.015,165.012,57.121,160.060
C08051=1015.687,-105.291,399.023,165.008,57.127,160.060
C08052=1015.682,-105.541,399.031,165.006,57.133,160.061
C08053=1015.677,-105.791,399.039,165.002,57.140,160.061
C08054=1015.673,-106.040,399.047,165.000,57.146,160.061
C08055=1015.668,-106.291,399.055,164.998,57.152,160.062
C08056=1015.662,-106.540,399.063,164.994,57.158,160.062
C08057=1015.658,-106.790,399.071,164.992,57.164,160.062
C08058=1015.653,-107.040,399.079,164.988,57.170,160.063
C08059=1015.648,-107.290,399.087,164.985,57.176,160.063
C08060=1015.643,-107.539,399.095,164.983,57.183,160.064
C08061=1015.638,-107.789,399.103,164.980,57.189,160.064
C08062=1015.633,-108.040,399.111,164.977,57.195,160.064
C08063=1015.629,-108.289,399.119,164.974,57.201,160.064
C08064=1015.624,-108.539,399.127,164.972,57.208,160.065
C08065=1015.619,-108.789,399.134,164.968,57.214,160.065
C08066=1015.614,-109.038,399.142,164.966,57.220,160.066
C08067=1015.609,-109.289,399.150,164.963,57.225,160.066
C08068=1015.604,-109.538,399.157,164.959,57.232,160.066
C08069=1015.599,-109.788,399.165,164.958,57.238,160.067
C08070=1015.594,-110.037,399.173,164.954,57.245,160.067
C08071=1015.589,-110.288,399.181,164.951,57.250,160.067
C08072=1015.585,-110.537,399.188,164.948,57.257,160.068
C08073=1015.580,-110.787,399.197,164.945,57.262,160.068
C08074=1015.575,-111.037,399.204,164.943,57.268,160.068
C08075=1015.570,-111.287,399.212,164.940,57.275,160.069
C08076=1015.565,-111.537,399.219,164.937,57.281,160.069
C08077=1015.560,-111.786,399.227,164.934,57.287,160.069
C08078=1015.555,-112.036,399.235,164.931,57.293,160.070
C08079=1015.551,-112.286,399.242,164.929,57.299,160.070
C08080=1015.546,-112.536,399.250,164.925,57.305,160.070
C08081=1015.541,-112.785,399.258,164.922,57.311,160.071
C08082=1015.536,-113.036,399.266,164.921,57.318,160.071
C08083=1015.532,-113.285,399.273,164.917,57.324,160.072
C08084=1015.526,-113.535,399.280,164.914,57.330,160.072
C08085=1015.522,-113.785,399.288,164.912,57.336,160.072
C08086=1015.516,-114.035,399.296,164.908,57.342,160.073
C08087=1015.512,-114.284,399.304,164.906,57.348,160.073
C08088=1015.507,-114.535,399.311,164.903,57.354,160.073
C08089=1015.503,-114.784,399.319,164.900,57.360,160.074
C08090=1015.497,-115.034,399.326,164.897,57.366,160.074
C08091=1015.493,-115.284,399.333,164.894,57.372,160.074
C08092=1015.488,-115.534,399.341,164.891,57.378,160.075
C08093=1015.483,-115.784,399.349,164.889,57.384,160.075
C08094=1015.479,-116.034,399.356,164.886,57.391,160.075
C08095=1015.473,-116.284,399.363,164.883,57.397,160.076
C08096=1015.469,-116.533,399.371,164.881,57.402,160.076
C08097=1015.464,-116.784,399.378,164.877,57.409,160.076
C08098=1015.460,-117.033,399.386,164.874,57.414,160.077
C08099=1015.454,-117.283,399.393,164.872,57.420,160.077
C08100=1015.450,-117.533,399.400,164.868,57.427,160.077
C08101=1015.445,-117.768,399.408,164.866,57.432,160.078
C08102=1015.441,-118.003,399.414,164.863,57.438,160.078
C08103=1015.436,-118.237,399.421,164.860,57.443,160.078
C08104=1015.432,-118.473,399.428,164.858,57.449,160.079
C08105=1015.427,-118.707,399.435,164.855,57.455,160.079
C08106=1015.422,-118.942,399.442,164.852,57.460,160.079
C08107=1015.418,-119.177,399.449,164.850,57.466,160.079
C08108=1015.413,-119.412,399.456,164.847,57.472,160.080
C08109=1015.408,-119.662,399.463,164.845,57.478,160.080
C08110=1015.404,-119.911,399.471,164.842,57.484,160.081
C08111=1015.399,-120.162,399.478,164.839,57.490,160.081
C08112=1015.394,-120.412,399.485,164.836,57.496,160.081
C08113=1015.390,-120.661,399.492,164.834,57.502,160.082
C08114=1015.385,-120.911,399.500,164.831,57.507,160.082
C08115=1015.380,-121.161,399.507,164.828,57.514,160.082
C08116=1015.375,-121.410,399.514,164.825,57.520,160.082
C08117=1015.370,-121.723,399.523,164.821,57.527,160.083
C08118=1015.364,-122.035,399.532,164.818,57.534,160.083
C08119=1015.358,-122.347,399.541,164.814,57.542,160.084
C08120=1015.352,-122.659,399.550,164.811,57.549,160.084
C08121=1015.347,-122.910,399.557,164.808,57.556,160.084
C08122=1015.342,-123.159,399.564,164.805,57.562,160.085
C08123=1015.337,-123.409,399.571,164.803,57.567,160.085
C08124=1015.333,-123.659,399.579,164.800,57.572,160.085
C08125=1015.327,-123.908,399.586,164.796,57.579,160.085
C08126=1015.323,-124.158,399.593,164.794,57.585,160.086
C08127=1015.319,-124.408,399.600,164.791,57.591,160.086
C08128=1015.313,-124.658,399.607,164.789,57.596,160.087
C08129=1015.309,-124.908,399.615,164.786,57.602,160.087
C08130=1015.304,-125.158,399.621,164.783,57.609,160.087
C08131=1015.300,-125.407,399.628,164.780,57.614,160.087
C08132=1015.294,-125.657,399.635,164.778,57.620,160.088
C08133=1015.290,-125.908,399.642,164.775,57.626,160.088
C08134=1015.285,-126.157,399.649,164.772,57.632,160.088
C08135=1015.281,-126.407,399.656,164.769,57.638,160.089
C08136=1015.276,-126.657,399.662,164.767,57.644,160.089
C08137=1015.271,-126.907,399.670,164.764,57.650,160.090
C08138=1015.266,-127.157,399.676,164.761,57.656,160.090
C08139=1015.262,-127.406,399.684,164.758,57.661,160.090
C08140=1015.257,-127.656,399.690,164.755,57.667,160.090
C08141=1015.253,-127.906,399.697,164.753,57.673,160.091
C08142=1015.247,-128.155,399.704,164.749,57.680,160.091
C08143=1015.243,-128.405,399.711,164.747,57.684,160.091
C08144=1015.239,-128.655,399.719,164.744,57.689,160.091
C08145=1015.236,-128.904,399.728,164.742,57.694,160.091
C08146=1015.232,-129.154,399.737,164.739,57.698,160.091
C08147=1015.229,-129.403,399.747,164.736,57.701,160.091
C08148=1015.226,-129.653,399.757,164.734,57.704,160.091
C08149=1015.224,-129.902,399.768,164.732,57.706,160.091
C08150=1015.222,-130.152,399.780,164.729,57.707,160.090
C08151=1015.221,-130.402,399.791,164.726,57.708,160.090
C08152=1015.220,-130.651,399.804,164.724,57.709,160.089
C08153=1015.219,-130.901,399.818,164.722,57.709,160.089
C08154=1015.219,-131.151,399.831,164.720,57.708,160.088
C08155=1015.219,-131.401,399.846,164.718,57.707,160.087
C08156=1015.219,-131.650,399.861,164.716,57.704,160.086
C08157=1015.220,-131.900,399.876,164.713,57.702,160.085
C08158=1015.221,-132.150,399.893,164.712,57.699,160.084
C08159=1015.223,-132.399,399.910,164.710,57.696,160.083
C08160=1015.224,-132.649,399.928,164.708,57.692,160.082
C08161=1015.227,-132.898,399.945,164.705,57.687,160.080
C08162=1015.229,-133.148,399.964,164.704,57.682,160.079
C08163=1015.232,-133.398,399.983,164.703,57.676,160.078
C08164=1015.235,-133.647,400.003,164.701,57.670,160.076
C08165=1014.993,-133.674,399.599,164.670,58.036,160.133
C08166=1014.990,-133.424,399.579,164.670,58.043,160.135
C08167=1014.987,-133.175,399.560,164.673,58.048,160.136
C08168=1014.984,-132.925,399.542,164.674,58.053,160.138
C08169=1014.982,-132.675,399.524,164.677,58.058,160.139
C08170=1014.980,-132.426,399.506,164.679,58.062,160.141
C08171=1014.979,-132.176,399.489,164.680,58.066,160.142
C08172=1014.978,-131.926,399.473,164.682,58.069,160.143
C08173=1014.977,-131.677,399.457,164.684,58.071,160.144
C08174=1014.977,-131.427,399.442,164.687,58.073,160.145
C08175=1014.976,-131.178,399.427,164.688,58.074,160.145
C08176=1014.976,-130.928,399.413,164.691,58.074,160.146
C08177=1014.977,-130.678,399.400,164.693,58.075,160.147
C08178=1014.979,-130.429,399.388,164.696,58.075,160.147
C08179=1014.980,-130.179,399.376,164.698,58.074,160.148
C08180=1014.981,-129.929,399.364,164.700,58.072,160.148
C08181=1014.984,-129.679,399.353,164.702,58.070,160.148
C08182=1014.987,-129.430,399.343,164.705,58.067,160.149
C08183=1014.989,-129.180,399.333,164.707,58.064,160.149
C08184=1014.992,-128.930,399.324,164.710,58.060,160.149
C08185=1014.996,-128.681,399.316,164.712,58.056,160.149
C08186=1015.001,-128.432,399.307,164.715,58.051,160.149
C08187=1015.005,-128.182,399.300,164.718,58.046,160.148
C08188=1015.009,-127.932,399.293,164.721,58.040,160.148
C08189=1015.014,-127.682,399.287,164.723,58.034,160.148
C08190=1015.019,-127.433,399.279,164.726,58.028,160.147
C08191=1015.023,-127.183,399.273,164.729,58.023,160.147
C08192=1015.028,-126.933,399.266,164.732,58.016,160.147
C08193=1015.033,-126.684,399.259,164.735,58.011,160.147
C08194=1015.038,-126.433,399.252,164.737,58.005,160.146
C08195=1015.043,-126.183,399.245,164.739,57.999,160.146
C08196=1015.047,-125.933,399.238,164.743,57.992,160.146
C08197=1015.052,-125.684,399.231,164.745,57.987,160.145
C08198=1015.056,-125.434,399.224,164.748,57.981,160.145
C08199=1015.062,-125.184,399.218,164.751,57.975,160.145
C08200=1015.066,-124.934,399.210,164.754,57.969,160.145
C08201=1015.071,-124.684,399.204,164.757,57.963,160.144
C08202=1015.075,-124.434,399.197,164.759,57.957,160.144
C08203=1015.079,-124.185,399.189,164.762,57.951,160.143
C08204=1015.085,-123.935,399.182,164.764,57.946,160.143
C08205=1015.089,-123.685,399.175,164.768,57.939,160.143
C08206=1015.094,-123.435,399.169,164.770,57.933,160.142
C08207=1015.099,-123.186,399.161,164.773,57.928,160.142
C08208=1015.104,-122.935,399.153,164.776,57.922,160.142
C08209=1015.108,-122.685,399.147,164.779,57.916,160.142
C08210=1015.113,-122.436,399.140,164.782,57.910,160.141
C08211=1015.117,-122.186,399.133,164.784,57.904,160.141
C08212=1015.123,-121.936,399.125,164.786,57.898,160.141
C08213=1015.127,-121.686,399.118,164.790,57.892,160.140
C08214=1015.131,-121.436,399.111,164.792,57.886,160.140
C08215=1015.137,-121.186,399.104,164.795,57.880,160.140
C08216=1015.141,-120.936,399.097,164.797,57.874,160.139
C08217=1015.146,-120.687,399.089,164.801,57.868,160.139
C08218=1015.151,-120.438,399.082,164.803,57.862,160.139
C08219=1015.156,-120.187,399.075,164.806,57.856,160.138
C08220=1015.160,-119.937,399.068,164.809,57.850,160.138
C08221=1015.165,-119.688,399.061,164.812,57.844,160.138
C08222=1015.170,-119.437,399.053,164.814,57.838,160.137
C08223=1015.174,-119.188,399.046,164.818,57.832,160.137
C08224=1015.178,-118.938,399.039,164.820,57.826,160.137
C08225=1015.184,-118.688,399.031,164.823,57.820,160.136
C08226=1015.189,-118.406,399.024,164.826,57.814,160.136
C08227=1015.195,-118.124,399.015,164.829,57.807,160.136
C08228=1015.200,-117.841,399.007,164.832,57.800,160.135
C08229=1015.206,-117.560,398.999,164.836,57.793,160.135
C08230=1015.210,-117.310,398.991,164.839,57.787,160.135
C08231=1015.215,-117.060,398.983,164.842,57.781,160.134
C08232=1015.219,-116.810,398.976,164.844,57.775,160.134
C08233=1015.224,-116.561,398.969,164.848,57.769,160.134
C08234=1015.229,-116.310,398.961,164.850,57.763,160.133
C08235=1015.234,-116.061,398.954,164.852,57.756,160.133
C08236=1015.239,-115.810,398.946,164.855,57.750,160.133
C08237=1015.244,-115.561,398.940,164.858,57.744,160.132
C08238=1015.249,-115.311,398.932,164.860,57.738,160.132
C08239=1015.253,-115.061,398.924,164.864,57.732,160.132
C08240=1015.257,-114.811,398.917,164.866,57.726,160.131
C08241=1015.263,-114.561,398.910,164.869,57.720,160.131
C08242=1015.267,-114.312,398.902,164.872,57.714,160.131
C08243=1015.272,-114.061,398.895,164.875,57.708,160.130
C08244=1015.277,-113.812,398.886,164.877,57.702,160.130
C08245=1015.282,-113.562,398.879,164.881,57.696,160.130
C08246=1015.286,-113.312,398.871,164.883,57.690,160.129
C08247=1015.291,-113.062,398.864,164.887,57.684,160.129
C08248=1015.296,-112.813,398.857,164.889,57.678,160.129
C08249=1015.301,-112.562,398.849,164.892,57.672,160.128
C08250=1015.306,-112.313,398.842,164.895,57.665,160.128
C08251=1015.311,-112.063,398.833,164.897,57.659,160.127
C08252=1015.315,-111.813,398.826,164.900,57.653,160.127
C08253=1015.320,-111.563,398.818,164.903,57.647,160.127
C08254=1015.325,-111.313,398.810,164.906,57.641,160.126
C08255=1015.330,-111.063,398.803,164.909,57.635,160.126
C08256=1015.335,-110.814,398.795,164.912,57.629,160.126
C08257=1015.340,-110.564,398.787,164.914,57.622,160.125
C08258=1015.344,-110.314,398.780,164.917,57.616,160.125
C08259=1015.349,-110.064,398.772,164.920,57.610,160.125
C08260=1015.354,-109.815,398.764,164.923,57.604,160.124
C08261=1015.359,-109.565,398.756,164.926,57.598,160.124
C08262=1015.365,-109.232,398.747,164.929,57.590,160.123
C08263=1015.371,-108.900,398.736,164.934,57.581,160.123
C08264=1015.378,-108.567,398.726,164.937,57.573,160.122
C08265=1015.385,-108.235,398.715,164.941,57.565,160.122
C08266=1015.390,-107.985,398.708,164.944,57.558,160.122
C08267=1015.394,-107.735,398.700,164.947,57.553,160.121
C08268=1015.399,-107.485,398.692,164.948,57.546,160.121
C08269=1015.404,-107.235,398.684,164.952,57.540,160.120
C08270=1015.409,-106.985,398.677,164.954,57.534,160.120
C08271=1015.414,-106.736,398.668,164.958,57.528,160.120
C08272=1015.418,-106.486,398.661,164.961,57.522,160.119
C08273=1015.424,-106.236,398.652,164.964,57.515,160.119
C08274=1015.429,-105.986,398.644,164.966,57.509,160.119
C08275=1015.433,-105.736,398.637,164.968,57.503,160.118
C08276=1015.438,-105.487,398.628,164.972,57.497,160.118
C08277=1015.442,-105.236,398.620,164.975,57.491,160.118
C08278=1015.447,-104.987,398.612,164.978,57.485,160.117
C08279=1015.452,-104.737,398.604,164.980,57.478,160.117
C08280=1015.457,-104.487,398.596,164.984,57.472,160.117
C08281=1015.462,-104.237,398.588,164.986,57.466,160.116
C08282=1015.467,-103.988,398.580,164.990,57.460,160.116
C08283=1015.472,-103.737,398.572,164.991,57.453,160.115
C08284=1015.477,-103.488,398.564,164.994,57.447,160.115
C08285=1015.482,-103.238,398.556,164.998,57.441,160.115
C08286=1015.486,-103.014,398.549,165.000,57.435,160.114
C08287=1015.490,-102.789,398.541,165.003,57.430,160.114
C08288=1015.494,-102.565,398.534,165.006,57.424,160.114
C08289=1015.499,-102.340,398.527,165.008,57.418,160.113
C08290=1015.503,-102.116,398.519,165.011,57.412,160.113
C08291=1015.508,-101.891,398.512,165.013,57.408,160.113
C08292=1015.512,-101.666,398.505,165.015,57.402,160.112
C08293=1015.517,-101.442,398.497,165.018,57.396,160.112
C08294=1015.522,-101.192,398.489,165.021,57.390,160.112
C08295=1015.526,-100.943,398.481,165.023,57.383,160.111
C08296=1015.532,-100.693,398.473,165.027,57.377,160.111
C08297=1015.537,-100.443,398.465,165.029,57.371,160.110
C08298=1015.542,-100.193,398.457,165.032,57.364,160.110
C08299=1015.546,-99.944,398.448,165.035,57.358,160.109
C08300=1015.551,-99.693,398.440,165.038,57.352,160.109
C08301=1015.556,-99.444,398.432,165.041,57.345,160.109
C08302=1015.561,-99.194,398.423,165.044,57.339,160.108
C08303=1015.566,-98.944,398.416,165.047,57.333,160.108
C08304=1015.571,-98.694,398.407,165.049,57.326,160.107
C08305=1015.576,-98.445,398.399,165.053,57.320,160.107
C08306=1015.581,-98.194,398.391,165.055,57.313,160.107
C08307=1015.586,-97.945,398.383,165.058,57.307,160.106
C08308=1015.590,-97.695,398.374,165.061,57.301,160.106
C08309=1015.595,-97.445,398.366,165.064,57.295,160.106
C08310=1015.600,-97.195,398.357,165.066,57.289,160.105
C08311=1015.605,-96.945,398.349,165.070,57.282,160.105
C08312=1015.610,-96.696,398.340,165.072,57.276,160.104
C08313=1015.615,-96.446,398.331,165.075,57.271,160.104
C08314=1015.620,-96.196,398.323,165.078,57.264,160.104
C08315=1015.624,-95.946,398.314,165.080,57.258,160.103
C08316=1015.629,-95.697,398.305,165.084,57.252,160.103
C08317=1015.634,-95.446,398.298,165.086,57.246,160.103
C08318=1015.639,-95.196,398.289,165.089,57.239,160.102
C08319=1015.644,-94.947,398.280,165.092,57.233,160.102
C08320=1015.649,-94.697,398.271,165.096,57.227,160.101
C08321=1015.654,-94.447,398.262,165.097,57.220,160.101
C08322=1015.659,-94.198,398.254,165.101,57.214,160.101
C08323=1015.663,-93.948,398.245,165.104,57.208,160.100
C08324=1015.668,-93.698,398.237,165.107,57.201,160.100
C08325=1015.674,-93.448,398.228,165.109,57.195,160.099
C08326=1015.678,-93.198,398.219,165.113,57.189,160.099
C08327=1015.683,-92.949,398.211,165.115,57.182,160.098
C08328=1015.688,-92.699,398.202,165.118,57.176,160.098
C08329=1015.693,-92.449,398.193,165.121,57.170,160.098
C08330=1015.698,-92.199,398.185,165.124,57.163,160.097
C08331=1015.703,-91.949,398.176,165.126,57.158,160.097
C08332=1015.708,-91.700,398.167,165.129,57.151,160.096
C08333=1015.713,-91.450,398.158,165.132,57.145,160.096
C08334=1015.718,-91.200,398.150,165.135,57.139,160.096
C08335=1015.723,-90.951,398.141,165.138,57.132,160.095
C08336=1015.727,-90.701,398.132,165.141,57.126,160.095
C08337=1015.733,-90.451,398.124,165.144,57.119,160.094
C08338=1015.737,-90.201,398.115,165.146,57.113,160.094
C08339=1015.742,-89.951,398.106,165.150,57.106,160.094
C08340=1015.748,-89.702,398.098,165.152,57.100,160.093
C08341=1015.752,-89.452,398.089,165.156,57.094,160.093
C08342=1015.757,-89.202,398.080,165.158,57.087,160.092
C08343=1015.762,-88.952,398.071,165.161,57.081,160.092
C08344=1015.767,-88.703,398.062,165.164,57.074,160.092
C08345=1015.773,-88.453,398.053,165.167,57.068,160.091
C08346=1015.777,-88.203,398.044,165.170,57.061,160.091
C08347=1015.783,-87.953,398.036,165.172,57.056,160.090
C08348=1015.787,-87.703,398.027,165.175,57.049,160.090
C08349=1015.792,-87.454,398.018,165.178,57.042,160.089
C08350=1015.797,-87.203,398.009,165.181,57.036,160.089
C08351=1015.803,-86.953,398.000,165.184,57.029,160.088
C08352=1015.808,-86.704,397.991,165.188,57.023,160.088
C08353=1015.813,-86.454,397.982,165.189,57.016,160.087
C08354=1015.818,-86.174,397.973,165.193,57.009,160.087
C08355=1015.824,-85.894,397.963,165.197,57.002,160.087
C08356=1015.830,-85.615,397.953,165.199,56.994,160.086
C08357=1015.836,-85.335,397.943,165.202,56.987,160.085
///RCONF 1,0,0,0,0,0,0,0,0,0,0,0,0,0,0,0,0,0,0,0,0,0,0,0
C08358=1015.840,-85.085,397.933,165.206,56.981,160.085
C08359=1015.846,-84.835,397.925,165.209,56.974,160.085
C08360=1015.851,-84.585,397.917,165.211,56.967,160.084
C08361=1015.856,-84.336,397.907,165.214,56.961,160.084
C08362=1015.861,-84.086,397.898,165.217,56.954,160.083
C08363=1015.865,-83.836,397.889,165.219,56.948,160.083
C08364=1015.871,-83.586,397.881,165.223,56.941,160.082
C08365=1015.876,-83.336,397.871,165.226,56.934,160.082
C08366=1015.881,-83.086,397.862,165.228,56.928,160.081
C08367=1015.887,-82.837,397.854,165.232,56.922,160.081
C08368=1015.891,-82.587,397.844,165.235,56.915,160.081
C08369=1015.897,-82.338,397.835,165.238,56.908,160.080
C08370=1015.901,-82.088,397.826,165.240,56.902,160.080
C08371=1015.907,-81.838,397.818,165.243,56.895,160.079
C08372=1015.912,-81.588,397.808,165.246,56.888,160.079
C08373=1015.917,-81.338,397.799,165.248,56.882,160.078
C08374=1015.923,-81.088,397.791,165.252,56.875,160.078
C08375=1015.927,-80.839,397.781,165.255,56.868,160.077
C08376=1015.933,-80.589,397.772,165.258,56.862,160.077
C08377=1015.938,-80.338,397.763,165.260,56.855,160.076
C08378=1015.943,-80.089,397.754,165.264,56.849,160.076
C08379=1015.948,-79.839,397.745,165.266,56.842,160.075
C08380=1015.953,-79.590,397.735,165.269,56.836,160.075
C08381=1015.957,-79.340,397.726,165.272,56.829,160.074
C08382=1015.963,-79.090,397.716,165.275,56.823,160.074
C08383=1015.968,-78.840,397.707,165.278,56.816,160.074
C08384=1015.973,-78.591,397.697,165.280,56.810,160.073
C08385=1015.978,-78.341,397.689,165.284,56.804,160.073
C08386=1015.983,-78.091,397.679,165.287,56.797,160.072
C08387=1015.988,-77.841,397.670,165.289,56.791,160.072
C08388=1015.994,-77.592,397.660,165.292,56.784,160.071
C08389=1015.998,-77.342,397.651,165.295,56.777,160.071
C08390=1016.003,-77.092,397.641,165.298,56.771,160.070
C08391=1016.008,-76.842,397.631,165.301,56.764,160.070
C08392=1016.014,-76.592,397.623,165.304,56.757,160.069
C08393=1016.018,-76.343,397.613,165.307,56.752,160.069
C08394=1016.024,-76.093,397.603,165.310,56.745,160.068
C08395=1016.029,-75.843,397.594,165.313,56.738,160.068
C08396=1016.034,-75.594,397.585,165.315,56.732,160.068
C08397=1016.039,-75.343,397.575,165.318,56.725,160.067
C08398=1016.044,-75.094,397.565,165.321,56.718,160.067
C08399=1016.049,-74.845,397.556,165.324,56.712,160.066
C08400=1016.054,-74.595,397.547,165.327,56.705,160.066
C08401=1016.059,-74.344,397.537,165.329,56.699,160.065
C08402=1016.064,-74.095,397.527,165.333,56.693,160.065
C08403=1016.069,-73.846,397.517,165.335,56.686,160.064
C08404=1016.074,-73.595,397.508,165.338,56.680,160.064
C08405=1016.079,-73.345,397.498,165.341,56.673,160.063
C08406=1016.084,-73.096,397.488,165.344,56.667,160.063
C08407=1016.089,-72.846,397.478,165.347,56.660,160.062
C08408=1016.094,-72.597,397.468,165.350,56.655,160.062
C08409=1016.100,-72.346,397.458,165.353,56.648,160.062
C08410=1016.104,-72.097,397.448,165.355,56.642,160.061
C08411=1016.109,-71.847,397.439,165.358,56.635,160.061
C08412=1016.114,-71.597,397.429,165.361,56.629,160.060
C08413=1016.119,-71.348,397.419,165.364,56.622,160.060
C08414=1016.124,-71.098,397.409,165.368,56.616,160.060
C08415=1016.129,-70.848,397.399,165.370,56.610,160.059
C08416=1016.134,-70.599,397.390,165.373,56.603,160.058
C08417=1016.140,-70.348,397.379,165.375,56.597,160.058
C08418=1016.145,-70.071,397.369,165.379,56.589,160.057
C08419=1016.150,-69.792,397.357,165.382,56.582,160.057
C08420=1016.156,-69.515,397.347,165.385,56.575,160.056
C08421=1016.162,-69.237,397.335,165.388,56.568,160.056
C08422=1016.167,-68.987,397.325,165.391,56.561,160.055
C08423=1016.172,-68.737,397.315,165.393,56.555,160.055
C08424=1016.177,-68.488,397.305,165.397,56.549,160.054
C08425=1016.182,-68.238,397.296,165.400,56.542,160.054
C08426=1016.187,-67.988,397.286,165.402,56.535,160.053
C08427=1016.192,-67.738,397.276,165.406,56.529,160.053
C08428=1016.197,-67.488,397.266,165.409,56.522,160.053
C08429=1016.202,-67.239,397.256,165.411,56.516,160.052
C08430=1016.208,-66.989,397.246,165.414,56.510,160.052
C08431=1016.212,-66.739,397.236,165.416,56.503,160.051
C08432=1016.218,-66.490,397.225,165.420,56.496,160.050
C08433=1016.223,-66.240,397.216,165.423,56.489,160.050
C08434=1016.228,-65.990,397.205,165.425,56.484,160.050
C08435=1016.233,-65.741,397.196,165.428,56.477,160.049
C08436=1016.239,-65.491,397.185,165.431,56.470,160.049
C08437=1016.244,-65.241,397.176,165.433,56.463,160.048
C08438=1016.249,-64.991,397.165,165.437,56.457,160.048
C08439=1016.253,-64.741,397.155,165.440,56.450,160.047
C08440=1016.259,-64.491,397.145,165.442,56.444,160.046
C08441=1016.263,-64.242,397.135,165.445,56.437,160.046
C08442=1016.269,-63.992,397.125,165.448,56.430,160.045
C08443=1016.274,-63.742,397.115,165.451,56.424,160.045
C08444=1016.279,-63.492,397.105,165.454,56.417,160.045
C08445=1016.285,-63.243,397.094,165.457,56.410,160.044
C08446=1016.290,-62.993,397.084,165.459,56.404,160.043
C08447=1016.295,-62.743,397.074,165.462,56.397,160.043
C08448=1016.300,-62.494,397.064,165.466,56.391,160.043
C08449=1016.305,-62.244,397.054,165.468,56.384,160.042
C08450=1016.310,-61.994,397.044,165.471,56.377,160.041
C08451=1016.316,-61.744,397.034,165.474,56.371,160.041
C08452=1016.321,-61.495,397.023,165.477,56.364,160.040
C08453=1016.326,-61.245,397.014,165.480,56.357,160.040
C08454=1016.332,-60.995,397.003,165.483,56.350,160.039
C08455=1016.336,-60.746,396.994,165.486,56.343,160.039
C08456=1016.342,-60.496,396.983,165.488,56.337,160.038
C08457=1016.348,-60.246,396.973,165.491,56.331,160.038
C08458=1016.352,-59.997,396.963,165.495,56.324,160.037
C08459=1016.358,-59.747,396.953,165.498,56.317,160.037
C08460=1016.363,-59.497,396.942,165.500,56.311,160.036
C08461=1016.367,-59.247,396.932,165.503,56.304,160.036
C08462=1016.373,-58.997,396.921,165.506,56.297,160.035
C08463=1016.378,-58.748,396.911,165.509,56.290,160.035
C08464=1016.383,-58.498,396.901,165.511,56.284,160.034
C08465=1016.389,-58.248,396.891,165.514,56.277,160.033
C08466=1016.394,-57.999,396.881,165.517,56.270,160.033
C08467=1016.399,-57.749,396.870,165.521,56.263,160.032
C08468=1016.405,-57.499,396.860,165.523,56.256,160.032
C08469=1016.411,-57.249,396.849,165.526,56.250,160.031
C08470=1016.415,-57.000,396.840,165.529,56.243,160.031
C08471=1016.421,-56.750,396.829,165.532,56.236,160.030
C08472=1016.426,-56.500,396.819,165.534,56.229,160.030
C08473=1016.431,-56.251,396.809,165.537,56.223,160.029
C08474=1016.437,-56.001,396.799,165.540,56.216,160.029
C08475=1016.442,-55.751,396.788,165.543,56.209,160.028
C08476=1016.448,-55.501,396.778,165.547,56.202,160.028
C08477=1016.452,-55.251,396.767,165.549,56.195,160.027
C08478=1016.458,-55.002,396.756,165.552,56.189,160.026
C08479=1016.463,-54.752,396.746,165.554,56.181,160.026
C08480=1016.468,-54.502,396.736,165.558,56.174,160.025
C08481=1016.474,-54.253,396.725,165.561,56.167,160.025
C08482=1016.480,-53.976,396.714,165.564,56.160,160.024
C08483=1016.486,-53.698,396.703,165.566,56.153,160.023
C08484=1016.492,-53.422,396.691,165.570,56.145,160.023
C08485=1016.498,-53.145,396.680,165.573,56.137,160.022
C08486=1016.503,-52.896,396.670,165.576,56.130,160.021
C08487=1016.509,-52.646,396.659,165.579,56.124,160.021
C08488=1016.514,-52.396,396.648,165.582,56.117,160.020
C08489=1016.519,-52.146,396.637,165.585,56.110,160.020
C08490=1016.525,-51.896,396.627,165.587,56.103,160.019
C08491=1016.530,-51.647,396.617,165.590,56.096,160.018
C08492=1016.535,-51.397,396.607,165.593,56.089,160.018
C08493=1016.541,-51.148,396.596,165.596,56.082,160.017
C08494=1016.546,-50.898,396.586,165.599,56.075,160.017
C08495=1016.551,-50.648,396.574,165.601,56.069,160.016
C08496=1016.557,-50.398,396.564,165.605,56.062,160.016
C08497=1016.562,-50.148,396.552,165.607,56.056,160.015
C08498=1016.567,-49.899,396.542,165.610,56.049,160.015
C08499=1016.572,-49.649,396.531,165.613,56.042,160.014
C08500=1016.577,-49.399,396.520,165.616,56.036,160.014
C08501=1016.582,-49.149,396.509,165.619,56.029,160.013
C08502=1016.588,-48.900,396.498,165.622,56.022,160.013
C08503=1016.593,-48.649,396.487,165.624,56.016,160.012
C08504=1016.599,-48.400,396.476,165.627,56.009,160.011
C08505=1016.603,-48.151,396.465,165.630,56.002,160.011
C08506=1016.609,-47.901,396.454,165.632,55.996,160.010
C08507=1016.613,-47.651,396.444,165.636,55.989,160.010
C08508=1016.619,-47.401,396.433,165.639,55.982,160.009
C08509=1016.624,-47.152,396.421,165.641,55.976,160.009
C08510=1016.630,-46.902,396.410,165.644,55.969,160.008
C08511=1016.635,-46.652,396.400,165.647,55.962,160.008
C08512=1016.640,-46.402,396.389,165.649,55.956,160.007
C08513=1016.645,-46.152,396.377,165.652,55.949,160.006
C08514=1016.651,-45.904,396.367,165.656,55.942,160.006
C08515=1016.656,-45.654,396.355,165.659,55.935,160.005
C08516=1016.661,-45.404,396.345,165.661,55.929,160.005
C08517=1016.666,-45.154,396.334,165.664,55.922,160.004
C08518=1016.672,-44.904,396.323,165.667,55.915,160.004
C08519=1016.677,-44.655,396.311,165.669,55.909,160.003
C08520=1016.682,-44.405,396.300,165.673,55.902,160.002
C08521=1016.687,-44.155,396.289,165.676,55.895,160.002
C08522=1016.693,-43.906,396.278,165.679,55.888,160.001
C08523=1016.698,-43.655,396.267,165.681,55.882,160.001
C08524=1016.704,-43.406,396.256,165.684,55.874,160.000
C08525=1016.709,-43.156,396.245,165.687,55.867,159.999
C08526=1016.714,-42.907,396.234,165.689,55.861,159.999
C08527=1016.719,-42.657,396.223,165.692,55.854,159.998
C08528=1016.725,-42.407,396.212,165.695,55.847,159.998
C08529=1016.730,-42.158,396.200,165.698,55.841,159.997
C08530=1016.736,-41.908,396.189,165.701,55.834,159.997
C08531=1016.741,-41.658,396.178,165.704,55.827,159.996
C08532=1016.747,-41.409,396.167,165.707,55.821,159.996
C08533=1016.752,-41.159,396.156,165.710,55.813,159.995
C08534=1016.757,-40.909,396.145,165.712,55.807,159.994
C08535=1016.762,-40.659,396.134,165.715,55.800,159.994
C08536=1016.768,-40.410,396.123,165.718,55.793,159.993
C08537=1016.773,-40.160,396.112,165.721,55.786,159.993
C08538=1016.778,-39.910,396.101,165.723,55.779,159.992
C08539=1016.783,-39.660,396.089,165.726,55.772,159.991
C08540=1016.789,-39.411,396.078,165.729,55.765,159.991
C08541=1016.794,-39.161,396.067,165.731,55.759,159.990
C08542=1016.800,-38.912,396.055,165.735,55.752,159.989
C08543=1016.805,-38.662,396.044,165.738,55.745,159.989
C08544=1016.810,-38.413,396.032,165.740,55.739,159.988
C08545=1016.815,-38.163,396.021,165.743,55.732,159.988
C08546=1016.821,-37.886,396.008,165.746,55.725,159.987
C08547=1016.827,-37.610,395.995,165.750,55.717,159.987
C08548=1016.833,-37.333,395.983,165.753,55.710,159.986
C08549=1016.839,-37.057,395.970,165.755,55.702,159.985
C08550=1016.844,-36.807,395.958,165.758,55.696,159.985
C08551=1016.849,-36.557,395.947,165.761,55.689,159.984
C08552=1016.855,-36.307,395.935,165.764,55.682,159.983
C08553=1016.860,-36.057,395.924,165.767,55.676,159.983
C08554=1016.866,-35.808,395.912,165.769,55.669,159.982
C08555=1016.871,-35.559,395.900,165.772,55.662,159.982
C08556=1016.876,-35.309,395.889,165.776,55.656,159.981
C08557=1016.881,-35.059,395.878,165.778,55.649,159.980
C08558=1016.887,-34.810,395.866,165.780,55.642,159.980
C08559=1016.892,-34.560,395.854,165.784,55.635,159.979
C08560=1016.897,-34.310,395.843,165.786,55.628,159.979
C08561=1016.902,-34.060,395.831,165.789,55.622,159.978
C08562=1016.908,-33.811,395.820,165.792,55.615,159.977
C08563=1016.913,-33.561,395.808,165.795,55.608,159.977
C08564=1016.918,-33.311,395.797,165.797,55.602,159.976
C08565=1016.923,-33.062,395.785,165.800,55.594,159.976
C08566=1016.929,-32.812,395.773,165.803,55.587,159.975
C08567=1016.935,-32.562,395.762,165.806,55.581,159.974
C08568=1016.940,-32.312,395.750,165.809,55.574,159.974
C08569=1016.945,-32.063,395.738,165.812,55.567,159.973
C08570=1016.950,-31.814,395.727,165.814,55.560,159.972
C08571=1016.957,-31.563,395.715,165.817,55.554,159.972
C08572=1016.962,-31.314,395.703,165.820,55.547,159.971
C08573=1016.967,-31.064,395.692,165.823,55.540,159.971
C08574=1016.972,-30.815,395.680,165.825,55.534,159.970
C08575=1016.977,-30.565,395.668,165.828,55.526,159.969
C08576=1016.984,-30.315,395.657,165.831,55.519,159.969
C08577=1016.989,-30.065,395.645,165.833,55.513,159.968
C08578=1016.994,-29.816,395.633,165.836,55.505,159.967
C08579=1016.999,-29.566,395.622,165.839,55.499,159.967
C08580=1017.005,-29.316,395.609,165.843,55.492,159.966
C08581=1017.011,-29.067,395.598,165.845,55.485,159.966
C08582=1017.016,-28.817,395.587,165.847,55.478,159.965
C08583=1017.021,-28.568,395.574,165.851,55.471,159.964
C08584=1017.026,-28.318,395.563,165.854,55.464,159.964
C08585=1017.032,-28.068,395.550,165.856,55.457,159.963
C08586=1017.038,-27.819,395.540,165.859,55.451,159.962
C08587=1017.043,-27.570,395.527,165.862,55.444,159.962
C08588=1017.048,-27.319,395.515,165.864,55.437,159.961
C08589=1017.053,-27.070,395.503,165.867,55.431,159.961
C08590=1017.058,-26.820,395.491,165.871,55.424,159.960
C08591=1017.064,-26.570,395.479,165.872,55.417,159.959
C08592=1017.069,-26.321,395.467,165.876,55.410,159.959
C08593=1017.074,-26.071,395.455,165.879,55.403,159.958
C08594=1017.080,-25.821,395.443,165.881,55.397,159.958
C08595=1017.085,-25.571,395.431,165.884,55.390,159.957
C08596=1017.090,-25.322,395.419,165.886,55.384,159.956
C08597=1017.096,-25.072,395.406,165.889,55.376,159.956
C08598=1017.101,-24.822,395.395,165.892,55.370,159.955
C08599=1017.107,-24.573,395.383,165.894,55.363,159.954
C08600=1017.113,-24.323,395.370,165.898,55.356,159.954
C08601=1017.117,-24.073,395.358,165.901,55.350,159.953
C08602=1017.122,-23.824,395.346,165.903,55.343,159.953
C08603=1017.128,-23.574,395.333,165.906,55.336,159.952
C08604=1017.133,-23.324,395.322,165.909,55.329,159.951
C08605=1017.138,-23.075,395.310,165.911,55.323,159.951
C08606=1017.144,-22.825,395.297,165.915,55.316,159.950
C08607=1017.150,-22.576,395.285,165.917,55.308,159.949
C08608=1017.155,-22.326,395.273,165.919,55.302,159.949
C08609=1017.160,-22.076,395.261,165.923,55.295,159.948
C08610=1017.166,-21.799,395.247,165.925,55.288,159.947
C08611=1017.172,-21.522,395.233,165.929,55.280,159.947
C08612=1017.178,-21.244,395.220,165.932,55.273,159.946
C08613=1017.184,-20.967,395.207,165.935,55.265,159.945
C08614=1017.190,-20.716,395.195,165.938,55.258,159.945
C08615=1017.195,-20.467,395.182,165.940,55.251,159.944
C08616=1017.200,-20.218,395.170,165.943,55.244,159.943
C08617=1017.206,-19.968,395.157,165.946,55.238,159.943
C08618=1017.211,-19.718,395.146,165.949,55.230,159.942
C08619=1017.217,-19.468,395.133,165.951,55.224,159.941
C08620=1017.222,-19.219,395.121,165.954,55.217,159.941
C08621=1017.228,-18.969,395.108,165.957,55.210,159.940
C08622=1017.233,-18.720,395.096,165.959,55.203,159.939
C08623=1017.239,-18.471,395.084,165.962,55.197,159.939
C08624=1017.244,-18.220,395.072,165.965,55.189,159.938
C08625=1017.249,-17.971,395.060,165.967,55.183,159.937
C08626=1017.255,-17.721,395.047,165.970,55.175,159.937
C08627=1017.260,-17.472,395.035,165.973,55.169,159.936
C08628=1017.266,-17.222,395.022,165.977,55.162,159.936
C08629=1017.271,-16.973,395.010,165.978,55.155,159.935
C08630=1017.277,-16.722,394.998,165.982,55.148,159.934
C08631=1017.282,-16.473,394.986,165.984,55.141,159.933
C08632=1017.288,-16.223,394.973,165.987,55.134,159.933
C08633=1017.293,-15.974,394.961,165.990,55.128,159.932
C08634=1017.298,-15.724,394.948,165.993,55.120,159.931
C08635=1017.304,-15.474,394.936,165.995,55.114,159.931
C08636=1017.310,-15.225,394.923,165.998,55.107,159.930
C08637=1017.314,-14.975,394.910,166.000,55.101,159.930
C08638=1017.320,-14.725,394.898,166.004,55.094,159.929
C08639=1017.325,-14.476,394.885,166.006,55.087,159.928
C08640=1017.331,-14.226,394.873,166.009,55.080,159.928
C08641=1017.336,-13.977,394.860,166.012,55.074,159.927
C08642=1017.341,-13.727,394.847,166.014,55.066,159.926
C08643=1017.347,-13.478,394.834,166.017,55.060,159.926
C08644=1017.353,-13.228,394.822,166.020,55.053,159.925
C08645=1017.357,-12.979,394.809,166.022,55.047,159.924
C08646=1017.363,-12.729,394.796,166.025,55.039,159.924
C08647=1017.368,-12.479,394.784,166.028,55.033,159.923
C08648=1017.374,-12.229,394.771,166.031,55.026,159.922
C08649=1017.379,-11.979,394.759,166.033,55.019,159.922
C08650=1017.384,-11.730,394.746,166.036,55.012,159.921
C08651=1017.390,-11.481,394.733,166.039,55.006,159.921
C08652=1017.395,-11.231,394.720,166.042,54.998,159.920
C08653=1017.401,-10.981,394.707,166.044,54.992,159.919
C08654=1017.406,-10.732,394.695,166.047,54.985,159.919
C08655=1017.411,-10.482,394.682,166.050,54.978,159.918
C08656=1017.417,-10.232,394.669,166.052,54.972,159.917
C08657=1017.422,-9.983,394.657,166.055,54.964,159.916
C08658=1017.428,-9.733,394.643,166.058,54.957,159.916
C08659=1017.433,-9.484,394.631,166.061,54.951,159.915
C08660=1017.438,-9.234,394.618,166.063,54.944,159.914
C08661=1017.444,-8.984,394.605,166.067,54.937,159.914
C08662=1017.450,-8.735,394.593,166.068,54.930,159.913
C08663=1017.455,-8.485,394.579,166.072,54.923,159.912
C08664=1017.461,-8.235,394.567,166.074,54.917,159.912
C08665=1017.465,-7.986,394.554,166.077,54.909,159.911
C08666=1017.471,-7.736,394.541,166.080,54.903,159.910
C08667=1017.477,-7.487,394.529,166.082,54.896,159.909
C08668=1017.482,-7.237,394.515,166.085,54.889,159.909
C08669=1017.488,-6.987,394.503,166.088,54.882,159.908
C08670=1017.493,-6.738,394.490,166.090,54.875,159.907
C08671=1017.499,-6.489,394.477,166.093,54.868,159.907
C08672=1017.505,-6.239,394.464,166.096,54.861,159.906
C08673=1017.509,-5.989,394.451,166.098,54.854,159.905
C08674=1017.516,-5.710,394.437,166.102,54.846,159.905
C08675=1017.522,-5.430,394.423,166.105,54.839,159.904
C08676=1017.529,-5.151,394.408,166.108,54.831,159.903
C08677=1017.534,-4.871,394.393,166.111,54.823,159.902
C08678=1017.540,-4.622,394.381,166.114,54.816,159.902
C08679=1017.546,-4.372,394.368,166.116,54.809,159.901
C08680=1017.551,-4.123,394.355,166.119,54.803,159.900
C08681=1017.556,-3.873,394.341,166.121,54.796,159.900
C08682=1017.561,-3.624,394.328,166.125,54.790,159.899
C08683=1017.566,-3.373,394.315,166.126,54.783,159.898
C08684=1017.573,-3.124,394.302,166.130,54.776,159.898
C08685=1017.578,-2.874,394.288,166.132,54.770,159.897
C08686=1017.583,-2.625,394.275,166.135,54.762,159.896
C08687=1017.588,-2.375,394.262,166.138,54.756,159.896
C08688=1017.594,-2.126,394.248,166.140,54.749,159.895
C08689=1017.599,-1.877,394.235,166.143,54.742,159.894
C08690=1017.604,-1.627,394.222,166.145,54.736,159.894
C08691=1017.610,-1.377,394.208,166.149,54.729,159.893
C08692=1017.615,-1.127,394.195,166.150,54.722,159.892
C08693=1017.620,-0.878,394.182,166.154,54.715,159.892
C08694=1017.626,-0.628,394.169,166.156,54.709,159.891
C08695=1017.631,-0.379,394.155,166.159,54.701,159.890
C08696=1017.637,-0.129,394.142,166.161,54.695,159.889
C08697=1017.642,0.120,394.129,166.164,54.689,159.889
C08698=1017.647,0.370,394.115,166.167,54.681,159.888
C08699=1017.652,0.620,394.102,166.170,54.675,159.887
C08700=1017.658,0.870,394.088,166.173,54.668,159.887
C08701=1017.664,1.119,394.075,166.175,54.661,159.886
C08702=1017.669,1.368,394.062,166.178,54.655,159.886
C08703=1017.674,1.618,394.048,166.180,54.648,159.885
C08704=1017.680,1.867,394.034,166.183,54.641,159.884
C08705=1017.686,2.117,394.022,166.186,54.634,159.884
C08706=1017.691,2.367,394.008,166.188,54.627,159.883
C08707=1017.696,2.616,393.994,166.192,54.621,159.882
C08708=1017.701,2.866,393.981,166.193,54.614,159.881
C08709=1017.707,3.116,393.967,166.197,54.607,159.881
C08710=1017.713,3.365,393.954,166.198,54.600,159.880
C08711=1017.718,3.615,393.941,166.202,54.593,159.879
C08712=1017.723,3.864,393.927,166.205,54.586,159.878
C08713=1017.728,4.113,393.913,166.207,54.580,159.878
C08714=1017.734,4.363,393.901,166.210,54.572,159.877
C08715=1017.740,4.613,393.887,166.212,54.566,159.876
C08716=1017.745,4.863,393.873,166.215,54.559,159.876
C08717=1017.751,5.112,393.859,166.218,54.552,159.875
C08718=1017.756,5.362,393.846,166.220,54.545,159.874
C08719=1017.761,5.611,393.833,166.223,54.538,159.874
C08720=1017.767,5.860,393.819,166.225,54.531,159.873
C08721=1017.772,6.110,393.806,166.229,54.525,159.872
C08722=1017.778,6.360,393.792,166.231,54.517,159.871
C08723=1017.783,6.610,393.779,166.234,54.511,159.871
C08724=1017.789,6.859,393.765,166.237,54.504,159.870
C08725=1017.795,7.109,393.751,166.239,54.497,159.869
C08726=1017.800,7.359,393.738,166.242,54.490,159.868
C08727=1017.805,7.608,393.724,166.245,54.483,159.868
C08728=1017.812,7.858,393.711,166.247,54.476,159.867
C08729=1017.816,8.107,393.698,166.250,54.469,159.866
C08730=1017.822,8.356,393.684,166.252,54.463,159.866
C08731=1017.827,8.606,393.671,166.255,54.455,159.865
C08732=1017.833,8.856,393.657,166.258,54.449,159.864
C08733=1017.839,9.105,393.643,166.260,54.442,159.863
C08734=1017.844,9.355,393.630,166.263,54.434,159.863
C08735=1017.850,9.604,393.616,166.266,54.428,159.862
C08736=1017.855,9.854,393.602,166.268,54.421,159.861
C08737=1017.861,10.103,393.588,166.271,54.414,159.861
C08738=1017.867,10.385,393.573,166.274,54.406,159.860
C08739=1017.873,10.666,393.558,166.278,54.398,159.859
C08740=1017.879,10.948,393.542,166.280,54.390,159.858
C08741=1017.885,11.229,393.527,166.283,54.383,159.857
C08742=1017.891,11.478,393.513,166.286,54.376,159.856
C08743=1017.896,11.728,393.500,166.289,54.368,159.856
C08744=1017.903,11.977,393.486,166.291,54.362,159.855
C08745=1017.908,12.227,393.472,166.294,54.355,159.854
C08746=1017.914,12.476,393.459,166.297,54.347,159.853
C08747=1017.919,12.726,393.445,166.299,54.341,159.853
C08748=1017.925,12.975,393.431,166.302,54.334,159.852
C08749=1017.930,13.225,393.418,166.305,54.326,159.851
C08750=1017.936,13.474,393.404,166.307,54.320,159.851
C08751=1017.941,13.724,393.389,166.310,54.313,159.850
C08752=1017.946,13.974,393.375,166.312,54.306,159.849
C08753=1017.952,14.223,393.362,166.315,54.299,159.848
C08754=1017.957,14.473,393.348,166.318,54.293,159.848
C08755=1017.963,14.722,393.334,166.320,54.286,159.847
C08756=1017.968,14.972,393.320,166.323,54.279,159.846
C08757=1017.974,15.222,393.306,166.326,54.272,159.845
C08758=1017.979,15.471,393.292,166.327,54.265,159.844
C08759=1017.985,15.721,393.278,166.331,54.258,159.844
C08760=1017.991,15.970,393.264,166.334,54.251,159.843
C08761=1017.997,16.220,393.250,166.336,54.245,159.843
C08762=1018.002,16.469,393.236,166.339,54.237,159.842
C08763=1018.007,16.719,393.221,166.341,54.231,159.841
C08764=1018.012,16.969,393.207,166.344,54.224,159.840
C08765=1018.018,17.219,393.193,166.346,54.217,159.839
C08766=1018.024,17.467,393.179,166.349,54.210,159.839
C08767=1018.029,17.717,393.165,166.351,54.203,159.838
C08768=1018.035,17.967,393.151,166.355,54.197,159.837
C08769=1018.040,18.216,393.137,166.358,54.189,159.837
C08770=1018.046,18.466,393.123,166.359,54.183,159.836
C08771=1018.051,18.715,393.110,166.363,54.176,159.835
C08772=1018.057,18.964,393.095,166.365,54.169,159.834
C08773=1018.062,19.214,393.081,166.368,54.162,159.834
C08774=1018.067,19.464,393.067,166.370,54.155,159.833
C08775=1018.073,19.713,393.052,166.373,54.148,159.832
C08776=1018.079,19.963,393.038,166.375,54.142,159.831
C08777=1018.084,20.213,393.023,166.378,54.135,159.831
C08778=1018.089,20.462,393.010,166.380,54.128,159.830
C08779=1018.095,20.711,392.995,166.383,54.121,159.829
C08780=1018.100,20.961,392.981,166.387,54.114,159.829
C08781=1018.105,21.211,392.967,166.389,54.108,159.828
C08782=1018.111,21.460,392.952,166.392,54.100,159.827
C08783=1018.116,21.709,392.938,166.394,54.094,159.826
C08784=1018.122,21.960,392.924,166.397,54.087,159.825
C08785=1018.127,22.209,392.909,166.399,54.080,159.825
C08786=1018.133,22.459,392.895,166.402,54.073,159.824
C08787=1018.139,22.707,392.880,166.404,54.066,159.823
C08788=1018.144,22.957,392.866,166.407,54.060,159.823
C08789=1018.149,23.207,392.852,166.409,54.053,159.822
C08790=1018.155,23.456,392.837,166.413,54.046,159.821
C08791=1018.161,23.706,392.823,166.414,54.039,159.820
C08792=1018.166,23.956,392.809,166.417,54.032,159.819
C08793=1018.171,24.205,392.794,166.421,54.025,159.819
C08794=1018.177,24.455,392.780,166.423,54.018,159.818
C08795=1018.183,24.704,392.766,166.426,54.011,159.817
C08796=1018.189,24.954,392.752,166.428,54.005,159.817
C08797=1018.194,25.203,392.736,166.431,53.998,159.816
C08798=1018.199,25.453,392.722,166.433,53.991,159.815
C08799=1018.205,25.702,392.709,166.436,53.984,159.814
C08800=1018.210,25.951,392.694,166.438,53.977,159.813
C08801=1018.216,26.202,392.679,166.441,53.970,159.813
C08802=1018.223,26.484,392.663,166.444,53.963,159.812
C08803=1018.228,26.767,392.646,166.447,53.954,159.811
C08804=1018.235,27.050,392.630,166.450,53.947,159.810
C08805=1018.240,27.333,392.613,166.453,53.939,159.809
C08806=1018.246,27.582,392.599,166.456,53.932,159.809
C08807=1018.251,27.832,392.584,166.458,53.925,159.808
C08808=1018.257,28.081,392.569,166.461,53.918,159.807
C08809=1018.262,28.331,392.555,166.464,53.912,159.806
C08810=1018.268,28.580,392.540,166.466,53.905,159.806
C08811=1018.273,28.829,392.525,166.468,53.898,159.805
C08812=1018.279,29.080,392.511,166.472,53.891,159.804
C08813=1018.284,29.329,392.496,166.474,53.884,159.803
C08814=1018.290,29.578,392.481,166.477,53.878,159.803
C08815=1018.295,29.828,392.467,166.479,53.871,159.802
C08816=1018.301,30.078,392.452,166.482,53.863,159.801
C08817=1018.306,30.327,392.437,166.484,53.857,159.800
C08818=1018.311,30.576,392.423,166.487,53.850,159.800
C08819=1018.317,30.826,392.408,166.489,53.843,159.799
C08820=1018.323,31.075,392.393,166.493,53.837,159.798
C08821=1018.328,31.325,392.378,166.495,53.830,159.797
C08822=1018.333,31.574,392.364,166.498,53.822,159.796
C08823=1018.338,31.823,392.348,166.500,53.816,159.796
C08824=1018.345,32.074,392.334,166.503,53.809,159.795
C08825=1018.350,32.323,392.319,166.505,53.802,159.794
C08826=1018.355,32.572,392.304,166.508,53.795,159.794
C08827=1018.361,32.822,392.289,166.510,53.789,159.793
C08828=1018.366,33.071,392.275,166.513,53.781,159.792
C08829=1018.372,33.321,392.260,166.516,53.775,159.791
C08830=1018.378,33.570,392.245,166.518,53.768,159.790
C08831=1018.383,33.820,392.230,166.520,53.761,159.790
C08832=1018.388,34.069,392.216,166.523,53.754,159.789
C08833=1018.394,34.319,392.200,166.526,53.748,159.788
C08834=1018.400,34.568,392.186,166.529,53.740,159.787
C08835=1018.405,34.817,392.171,166.531,53.733,159.786
C08836=1018.411,35.068,392.156,166.534,53.727,159.786
C08837=1018.416,35.317,392.141,166.536,53.720,159.785
C08838=1018.422,35.566,392.127,166.539,53.713,159.784
C08839=1018.427,35.816,392.111,166.542,53.705,159.783
C08840=1018.433,36.065,392.097,166.544,53.699,159.783
C08841=1018.438,36.315,392.082,166.547,53.692,159.782
C08842=1018.444,36.564,392.067,166.549,53.685,159.781
C08843=1018.449,36.814,392.052,166.552,53.678,159.780
C08844=1018.455,37.064,392.036,166.555,53.672,159.780
C08845=1018.460,37.313,392.021,166.558,53.664,159.779
C08846=1018.465,37.554,392.006,166.560,53.658,159.778
C08847=1018.470,37.795,391.992,166.562,53.651,159.777
C08848=1018.475,38.036,391.978,166.564,53.645,159.777
C08849=1018.481,38.277,391.963,166.567,53.638,159.776
C08850=1018.487,38.518,391.949,166.570,53.632,159.775
C08851=1018.492,38.759,391.934,166.572,53.626,159.774
C08852=1018.498,39.000,391.919,166.574,53.619,159.774
C08853=1018.502,39.242,391.905,166.578,53.612,159.773
C08854=1018.508,39.491,391.890,166.580,53.605,159.772
C08855=1018.513,39.740,391.874,166.583,53.598,159.771
C08856=1018.519,39.990,391.859,166.585,53.592,159.771
C08857=1018.524,40.239,391.844,166.588,53.585,159.770
C08858=1018.530,40.489,391.829,166.590,53.578,159.769
C08859=1018.535,40.738,391.813,166.593,53.571,159.768
C08860=1018.540,40.988,391.798,166.595,53.564,159.768
C08861=1018.546,41.237,391.783,166.598,53.557,159.767
C08862=1018.551,41.486,391.767,166.600,53.550,159.766
C08863=1018.557,41.736,391.752,166.604,53.544,159.765
C08864=1018.562,41.985,391.737,166.606,53.537,159.764
C08865=1018.569,42.235,391.722,166.609,53.530,159.764
C08866=1018.575,42.535,391.703,166.611,53.522,159.763
C08867=1018.581,42.835,391.685,166.615,53.513,159.762
C08868=1018.587,43.135,391.666,166.618,53.506,159.761
C08869=1018.594,43.434,391.647,166.622,53.498,159.760
C08870=1018.599,43.683,391.632,166.623,53.491,159.759
C08871=1018.604,43.932,391.617,166.625,53.484,159.758
C08872=1018.610,44.182,391.601,166.629,53.478,159.758
C08873=1018.615,44.431,391.585,166.631,53.471,159.757
C08874=1018.621,44.681,391.570,166.634,53.464,159.756
C08875=1018.626,44.930,391.555,166.636,53.457,159.756
C08876=1018.632,45.180,391.539,166.639,53.451,159.755
C08877=1018.636,45.429,391.523,166.642,53.444,159.754
C08878=1018.642,45.679,391.507,166.644,53.437,159.753
C08879=1018.647,45.928,391.492,166.647,53.431,159.753
C08880=1018.653,46.178,391.476,166.649,53.424,159.752
C08881=1018.658,46.427,391.461,166.651,53.417,159.751
C08882=1018.663,46.677,391.445,166.655,53.411,159.750
C08883=1018.669,46.926,391.430,166.657,53.404,159.749
C08884=1018.674,47.176,391.414,166.660,53.397,159.749
C08885=1018.680,47.425,391.398,166.662,53.390,159.748
C08886=1018.685,47.675,391.383,166.665,53.383,159.747
C08887=1018.691,47.923,391.367,166.667,53.376,159.746
C08888=1018.696,48.173,391.351,166.670,53.370,159.746
C08889=1018.701,48.423,391.336,166.673,53.363,159.745
C08890=1018.707,48.672,391.320,166.675,53.356,159.744
C08891=1018.712,48.921,391.305,166.678,53.350,159.743
C08892=1018.717,49.172,391.289,166.680,53.343,159.742
C08893=1018.722,49.420,391.273,166.683,53.336,159.742
C08894=1018.728,49.670,391.257,166.686,53.329,159.741
C08895=1018.733,49.919,391.242,166.688,53.323,159.740
C08896=1018.739,50.169,391.226,166.691,53.315,159.739
C08897=1018.745,50.419,391.210,166.693,53.309,159.738
C08898=1018.750,50.667,391.194,166.696,53.302,159.738
C08899=1018.756,50.917,391.179,166.698,53.295,159.737
C08900=1018.761,51.167,391.164,166.701,53.288,159.736
C08901=1018.767,51.416,391.147,166.703,53.281,159.735
C08902=1018.772,51.665,391.132,166.707,53.275,159.735
C08903=1018.778,51.915,391.116,166.709,53.268,159.734
C08904=1018.783,52.165,391.100,166.712,53.261,159.733
C08905=1018.788,52.414,391.085,166.714,53.254,159.732
C08906=1018.794,52.663,391.068,166.717,53.247,159.732
C08907=1018.799,52.913,391.053,166.719,53.241,159.731
C08908=1018.805,53.162,391.037,166.722,53.233,159.730
C08909=1018.810,53.412,391.021,166.724,53.227,159.729
C08910=1018.816,53.661,391.006,166.726,53.220,159.728
C08911=1018.821,53.911,390.990,166.730,53.213,159.728
C08912=1018.827,54.159,390.974,166.732,53.206,159.727
C08913=1018.832,54.409,390.959,166.735,53.199,159.726
C08914=1018.838,54.659,390.942,166.737,53.192,159.725
C08915=1018.843,54.908,390.927,166.740,53.185,159.724
C08916=1018.849,55.157,390.911,166.742,53.178,159.723
C08917=1018.855,55.407,390.895,166.745,53.172,159.723
C08918=1018.860,55.656,390.879,166.747,53.165,159.722
C08919=1018.865,55.906,390.863,166.751,53.158,159.721
C08920=1018.871,56.155,390.847,166.753,53.151,159.720
C08921=1018.876,56.405,390.832,166.756,53.144,159.720
C08922=1018.882,56.654,390.816,166.758,53.137,159.719
C08923=1018.888,56.904,390.800,166.761,53.130,159.718
C08924=1018.893,57.153,390.784,166.763,53.124,159.717
C08925=1018.899,57.403,390.769,166.766,53.117,159.716
C08926=1018.905,57.652,390.752,166.769,53.110,159.716
C08927=1018.910,57.901,390.737,166.771,53.103,159.715
C08928=1018.916,58.151,390.721,166.774,53.096,159.714
C08929=1018.921,58.401,390.705,166.776,53.089,159.713
C08930=1018.927,58.683,390.687,166.779,53.081,159.712
C08931=1018.934,58.966,390.669,166.783,53.073,159.711
C08932=1018.940,59.248,390.651,166.786,53.065,159.710
C08933=1018.946,59.531,390.633,166.788,53.058,159.709
C08934=1018.952,59.781,390.617,166.792,53.050,159.709
C08935=1018.957,60.031,390.601,166.794,53.044,159.708
C08936=1018.963,60.279,390.585,166.797,53.036,159.707
C08937=1018.969,60.529,390.569,166.799,53.030,159.706
C08938=1018.974,60.779,390.553,166.802,53.022,159.705
C08939=1018.980,61.027,390.538,166.804,53.016,159.704
C08940=1018.986,61.276,390.521,166.807,53.009,159.704
C08941=1018.991,61.526,390.506,166.810,53.001,159.703
C08942=1018.997,61.776,390.489,166.812,52.995,159.702
C08943=1019.002,62.025,390.474,166.815,52.987,159.701
C08944=1019.007,62.275,390.457,166.817,52.981,159.700
C08945=1019.013,62.524,390.441,166.820,52.973,159.700
C08946=1019.019,62.774,390.426,166.822,52.967,159.699
C08947=1019.025,63.023,390.409,166.825,52.960,159.698
C08948=1019.030,63.272,390.393,166.827,52.953,159.697
C08949=1019.036,63.522,390.377,166.831,52.946,159.697
C08950=1019.042,63.771,390.360,166.833,52.939,159.696
C08951=1019.046,64.021,390.344,166.836,52.932,159.695
C08952=1019.052,64.270,390.328,166.838,52.926,159.694
C08953=1019.057,64.520,390.312,166.841,52.918,159.693
C08954=1019.063,64.769,390.295,166.844,52.912,159.693
C08955=1019.069,65.018,390.279,166.847,52.905,159.692
C08956=1019.074,65.268,390.262,166.849,52.898,159.691
C08957=1019.079,65.517,390.246,166.852,52.891,159.690
C08958=1019.084,65.767,390.230,166.854,52.884,159.689
C08959=1019.090,66.016,390.214,166.856,52.878,159.688
C08960=1019.096,66.266,390.197,166.859,52.871,159.688
C08961=1019.101,66.515,390.181,166.862,52.865,159.687
C08962=1019.106,66.764,390.164,166.865,52.857,159.686
C08963=1019.112,67.014,390.148,166.867,52.851,159.685
C08964=1019.118,67.263,390.132,166.870,52.843,159.684
C08965=1019.123,67.513,390.115,166.872,52.837,159.684
C08966=1019.129,67.762,390.099,166.875,52.830,159.683
C08967=1019.134,68.011,390.082,166.877,52.823,159.682
C08968=1019.140,68.260,390.066,166.881,52.816,159.681
C08969=1019.145,68.510,390.049,166.883,52.810,159.680
C08970=1019.150,68.760,390.032,166.886,52.802,159.680
C08971=1019.156,69.009,390.016,166.888,52.796,159.679
C08972=1019.161,69.259,389.999,166.890,52.789,159.678
C08973=1019.167,69.507,389.983,166.894,52.782,159.677
C08974=1019.172,69.757,389.966,166.896,52.776,159.676
C08975=1019.177,70.007,389.950,166.899,52.769,159.676
C08976=1019.183,70.256,389.933,166.901,52.762,159.675
C08977=1019.188,70.506,389.916,166.904,52.755,159.674
C08978=1019.194,70.755,389.900,166.906,52.748,159.673
C08979=1019.199,71.005,389.883,166.910,52.742,159.673
C08980=1019.204,71.254,389.867,166.912,52.735,159.672
C08981=1019.210,71.502,389.850,166.914,52.728,159.671
C08982=1019.216,71.752,389.833,166.917,52.721,159.670
C08983=1019.221,72.002,389.816,166.919,52.714,159.669
C08984=1019.227,72.251,389.800,166.922,52.707,159.668
C08985=1019.232,72.501,389.783,166.925,52.701,159.668
C08986=1019.238,72.750,389.767,166.928,52.694,159.667
C08987=1019.243,73.000,389.750,166.930,52.687,159.666
C08988=1019.248,73.249,389.733,166.933,52.680,159.665
C08989=1019.254,73.497,389.716,166.935,52.673,159.664
C08990=1019.259,73.747,389.700,166.939,52.666,159.664
C08991=1019.264,73.997,389.683,166.941,52.659,159.663
C08992=1019.270,74.246,389.667,166.944,52.653,159.662
C08993=1019.276,74.496,389.650,166.946,52.646,159.661
C08994=1019.282,74.778,389.631,166.949,52.638,159.660
C08995=1019.288,75.061,389.611,166.952,52.631,159.659
C08996=1019.294,75.343,389.592,166.956,52.622,159.658
C08997=1019.300,75.626,389.573,166.958,52.615,159.657
C08998=1019.306,75.875,389.557,166.960,52.608,159.657
C08999=1019.311,76.125,389.540,166.964,52.601,159.656
C09000=1019.317,76.374,389.523,166.966,52.595,159.655
C09001=1019.322,76.623,389.506,166.969,52.588,159.654
C09002=1019.328,76.873,389.490,166.971,52.581,159.653
C09003=1019.333,77.122,389.472,166.974,52.574,159.653
C09004=1019.339,77.371,389.455,166.977,52.567,159.652
C09005=1019.344,77.621,389.438,166.979,52.560,159.651
C09006=1019.349,77.870,389.421,166.982,52.554,159.650
C09007=1019.355,78.120,389.404,166.984,52.547,159.649
C09008=1019.360,78.369,389.387,166.988,52.540,159.649
C09009=1019.365,78.619,389.370,166.990,52.533,159.648
C09010=1019.371,78.868,389.353,166.993,52.527,159.647
C09011=1019.376,79.117,389.335,166.995,52.520,159.646
C09012=1019.381,79.367,389.318,166.998,52.514,159.645
C09013=1019.388,79.616,389.301,167.001,52.506,159.645
C09014=1019.393,79.865,389.284,167.003,52.500,159.644
C09015=1019.398,80.115,389.268,167.006,52.493,159.643
C09016=1019.403,80.364,389.250,167.009,52.487,159.642
C09017=1019.408,80.613,389.234,167.012,52.480,159.642
C09018=1019.414,80.862,389.216,167.014,52.473,159.641
C09019=1019.419,81.112,389.199,167.016,52.466,159.640
C09020=1019.424,81.361,389.182,167.019,52.459,159.639
C09021=1019.430,81.610,389.165,167.021,52.452,159.638
C09022=1019.436,81.860,389.147,167.025,52.446,159.638
C09023=1019.441,82.110,389.130,167.027,52.439,159.637
C09024=1019.446,82.359,389.112,167.030,52.432,159.636
C09025=1019.452,82.608,389.095,167.032,52.425,159.635
C09026=1019.457,82.857,389.078,167.036,52.418,159.634
C09027=1019.462,83.107,389.061,167.038,52.412,159.633
C09028=1019.468,83.356,389.044,167.041,52.404,159.633
C09029=1019.473,83.606,389.027,167.043,52.398,159.632
C09030=1019.479,83.855,389.009,167.047,52.391,159.631
C09031=1019.485,84.104,388.993,167.049,52.385,159.630
C09032=1019.490,84.353,388.975,167.051,52.378,159.629
C09033=1019.495,84.603,388.958,167.054,52.371,159.629
C09034=1019.501,84.852,388.941,167.056,52.364,159.628
C09035=1019.506,85.102,388.924,167.059,52.357,159.627
C09036=1019.512,85.351,388.906,167.062,52.350,159.626
C09037=1019.517,85.600,388.889,167.065,52.343,159.625
C09038=1019.522,85.849,388.872,167.067,52.337,159.624
C09039=1019.528,86.098,388.854,167.070,52.330,159.624
C09040=1019.533,86.348,388.838,167.072,52.323,159.623
C09041=1019.539,86.597,388.820,167.075,52.316,159.622
C09042=1019.545,86.847,388.802,167.078,52.309,159.621
C09043=1019.550,87.096,388.785,167.081,52.302,159.620
C09044=1019.555,87.346,388.768,167.083,52.295,159.619
C09045=1019.561,87.595,388.751,167.086,52.288,159.619
C09046=1019.566,87.844,388.733,167.088,52.282,159.618
C09047=1019.572,88.093,388.716,167.092,52.275,159.617
C09048=1019.577,88.343,388.699,167.095,52.267,159.616
C09049=1019.582,88.592,388.681,167.097,52.261,159.615
C09050=1019.588,88.841,388.664,167.100,52.254,159.615
C09051=1019.594,89.091,388.646,167.103,52.248,159.614
C09052=1019.599,89.340,388.629,167.106,52.241,159.613
C09053=1019.605,89.589,388.611,167.108,52.234,159.612
C09054=1019.610,89.838,388.594,167.110,52.227,159.611
C09055=1019.615,90.088,388.576,167.113,52.220,159.611
C09056=1019.620,90.337,388.559,167.116,52.214,159.610
C09057=1019.626,90.587,388.541,167.119,52.207,159.609
C09058=1019.632,90.870,388.521,167.122,52.199,159.608
C09059=1019.638,91.152,388.500,167.125,52.192,159.607
C09060=1019.644,91.435,388.481,167.128,52.184,159.606
C09061=1019.650,91.718,388.461,167.131,52.177,159.605
C09062=1019.655,91.967,388.443,167.134,52.170,159.605
C09063=1019.661,92.216,388.426,167.136,52.163,159.604
C09064=1019.666,92.466,388.407,167.139,52.156,159.603
C09065=1019.672,92.715,388.390,167.142,52.150,159.602
C09066=1019.677,92.964,388.372,167.145,52.142,159.601
C09067=1019.682,93.213,388.354,167.147,52.136,159.601
C09068=1019.687,93.463,388.337,167.150,52.129,159.600
C09069=1019.693,93.712,388.320,167.152,52.122,159.599
C09070=1019.699,93.962,388.302,167.156,52.116,159.598
C09071=1019.704,94.211,388.284,167.158,52.109,159.597
C09072=1019.709,94.460,388.266,167.161,52.102,159.597
C09073=1019.715,94.709,388.248,167.164,52.095,159.596
C09074=1019.720,94.958,388.231,167.167,52.088,159.595
C09075=1019.726,95.208,388.212,167.169,52.082,159.594
C09076=1019.731,95.457,388.195,167.172,52.075,159.593
C09077=1019.737,95.706,388.177,167.174,52.068,159.592
C09078=1019.742,95.956,388.159,167.178,52.061,159.592
C09079=1019.747,96.205,388.141,167.180,52.054,159.591
C09080=1019.753,96.454,388.124,167.183,52.047,159.590
C09081=1019.759,96.703,388.106,167.185,52.041,159.589
C09082=1019.763,96.953,388.088,167.189,52.034,159.588
C09083=1019.769,97.202,388.070,167.191,52.027,159.587
C09084=1019.775,97.452,388.052,167.194,52.020,159.587
C09085=1019.781,97.701,388.035,167.196,52.013,159.586
C09086=1019.785,97.950,388.017,167.199,52.006,159.585
C09087=1019.791,98.199,387.999,167.202,52.000,159.584
C09088=1019.797,98.449,387.981,167.205,51.993,159.583
C09089=1019.802,98.698,387.963,167.207,51.986,159.583
C09090=1019.807,98.947,387.945,167.210,51.979,159.582
C09091=1019.813,99.196,387.928,167.214,51.972,159.581
C09092=1019.818,99.446,387.909,167.216,51.965,159.580
C09093=1019.824,99.695,387.892,167.218,51.959,159.579
C09094=1019.829,99.945,387.874,167.222,51.952,159.579
C09095=1019.835,100.194,387.856,167.224,51.946,159.578
C09096=1019.840,100.443,387.837,167.227,51.939,159.577
C09097=1019.845,100.692,387.819,167.229,51.932,159.576
C09098=1019.850,100.942,387.801,167.233,51.925,159.575
C09099=1019.855,101.192,387.782,167.235,51.918,159.574
